RoboDK station: kr30 cnc template amana 46348 - paulina NEW THING 2.rdk

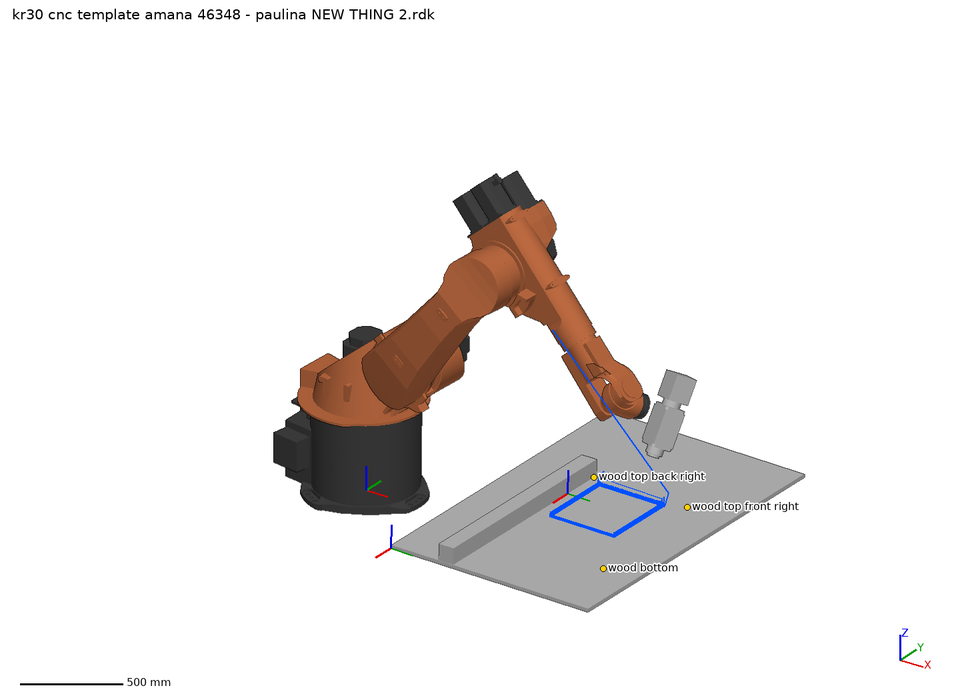
[picture v0: the station drawn from its stored meshes, robots at their saved joint values, targets as dots, program paths as lines]
Station kr30 cnc template amana 46348 - paulina NEW THING 2. Poses are relative to the parent item; angles as X-Y-Z fixed-axis rotations.
  - frame KUKA KR 30 HA Base at (0, 0, 0) mm
    - robot KUKA KR 30 HA: 6 axes, payload 30 kg, reach 2033 mm, repeatability 0.05 mm, weight 665 kg
        modified DH rows (alpha deg, a mm, theta deg, d mm): 0, 0, 0, 815; -90, 350, 0, 0; 0, 850, -90, 0; -90, 145, 0, 820; 90, 0, 0, 0; -90, 0, 180, 170
        joint limits [-185, -135, -120, -350, -119, -350] to [185, 35, 158, 350, 119, 350]; home [0, -90, 90, 0, 0, 0]; saved at [2.902, -51.207, 99.996, 272.3, 54.468, -220.075]
      - tool rc90 spindle mm, TCP at (267.95, 0.68, 160.99) mm, rotated rx 0 ry 90 rz 0 deg, size 110 x 421.3 x 118 mm, geometry from rc90 spindle mm.stl
    - frame Tabletop at (921.82, -1104.91, 385) mm, rotated rx -0.93 ry -0.21 rz -89.9 deg
      - object tabletop CHECK HEIGHT at (-1839.9, 0, 0) mm, size 1839.9 x 1168.4 x 19 mm, geometry from kr30 tabletop mm.stl
      - object kr30 pipe jig base at (-1220, -610.6, 0) mm, size 1217.6 x 88.9 x 88.9 mm, geometry from kr30 pipe jig base.stl
      - frame Frame 3 at (-930, 400, 45) mm
      - target wood top back right (Cartesian target) at (-1141.49, 406.84, 52.26) mm, rotated rx 18.07 ry 89.88 rz 108.17 deg; joints [-2.086, -55.392, 143.759, 178.106, 87.553, -179.775] of KUKA KR 30 HA
      - target wood bottom (Cartesian target) at (-376.62, 995.52, 35.89) mm, rotated rx 18.07 ry 89.88 rz 108.17 deg; joints [24.587, -27.296, 76.752, 211.623, 53.064, -199.759] of KUKA KR 30 HA
      - target wood top front right (Cartesian target) at (-1142.68, 960.22, 52.55) mm, rotated rx 18.06 ry 89.88 rz 108.16 deg; joints [-1.42, -37.516, 98.016, 178.579, 59.693, -179.129] of KUKA KR 30 HA
  - machining project Machining Settings: C:/Users/Research Office/Desktop/paulina a5.apt | rotZ(0) | rotX(0)*rotY(0) | rotZ(0)
  - program Machining (2349 instructions, listed below)
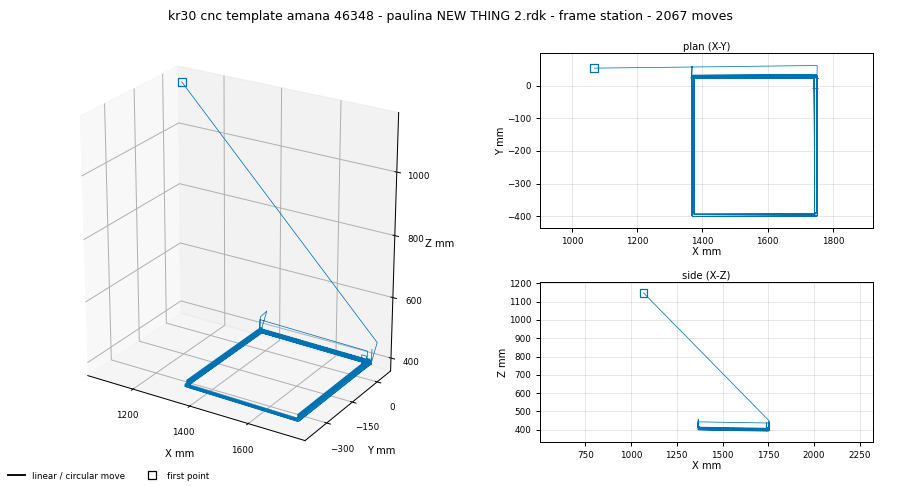
[picture p0: tool path of kr30 cnc template amana 46348 - paulina NEW THING 2.rdk in frame station, 2067 of 2067 moves have a stored position in this frame; points joined in program order, loops and branches not executed]

--- program Machining (robot KUKA KR 30 HA) ---
  Smooth(10)
  Print: /'1001'
  Print: /''
  Print: /'diagonal cut'
  Set speed (100.0 mm/s)
  Set Ref.: Frame 3
  Set Tool: rc90 spindle mm
  Show rc90 spindle mm
  MoveJ 1 to (-225.94, -263.82, 724.05) mm, rotated rx -179.73 ry 3.45 rz -91.41 deg; joints [-5.005, -121.314, 141.062, 163.754, 23.118, -164.211]
  MoveL 2 to (-235.36, 431, 39.15) mm, rotated rx -174.06 ry -29.54 rz -11.91 deg; joints [2.832, -37.469, 83.05, -73.25, 63.513, 134.274]
  MoveL 3 to (-235.36, 431, 39.15) mm, rotated rx -174.06 ry -29.54 rz -11.91 deg; joints [2.832, -37.469, 83.05, -73.25, 63.513, 134.274]
  Set speed (100.0 mm/s)
  MoveL 4 to (-206.65, 431, -10.41) mm, rotated rx -174.06 ry -29.54 rz -11.91 deg; joints [3.804, -35.34, 82.979, -73.62, 63.566, 136.691]
  Set speed (38.1 mm/s)
  MoveL 5 to (-201.55, 431, -19.21) mm, rotated rx -174.06 ry -29.54 rz -11.91 deg; joints [3.976, -34.949, 82.939, -73.676, 63.579, 137.104]
  MoveL 6 to (-200.68, 431, -19.44) mm, rotated rx -174.06 ry -29.54 rz -11.91 deg; joints [4.005, -34.936, 82.932, -73.66, 63.596, 137.117]
  Set speed (76.2 mm/s)
  MoveL 7 to (-202.44, 431, -12.48) mm, rotated rx -174.06 ry -29.54 rz -11.91 deg; joints [3.945, -35.237, 82.947, -73.562, 63.638, 136.796]
  MoveL 8 to (-201.13, 431, -12.23) mm, rotated rx -174.06 ry -29.54 rz -11.91 deg; joints [3.989, -35.243, 82.936, -73.526, 63.671, 136.788]
  MoveL 9 to (-196.56, 431, -16.91) mm, rotated rx -174.06 ry -29.54 rz -11.91 deg; joints [4.143, -35.027, 82.898, -73.511, 63.72, 137.012]
  Set speed (38.1 mm/s)
  MoveL 10 to (-196.33, 431, -16.04) mm, rotated rx -174.06 ry -29.54 rz -11.91 deg; joints [4.151, -35.063, 82.897, -73.488, 63.735, 136.973]
  Set speed (100.0 mm/s)
  MoveL 11 to (-203.65, 431, -3.41) mm, rotated rx -174.06 ry -29.54 rz -11.91 deg; joints [3.903, -35.623, 82.951, -73.408, 63.719, 136.379]
  MoveL 12 to (-199.05, 427.82, -0.75) mm, rotated rx -174.06 ry -29.54 rz -11.91 deg; joints [4.065, -35.896, 83.273, -73.328, 63.81, 136.466]
  Set speed (38.1 mm/s)
  MoveL 13 to (-197.47, 427.82, -3.47) mm, rotated rx -174.06 ry -29.54 rz -11.91 deg; joints [4.118, -35.776, 83.262, -73.346, 63.813, 136.595]
  MoveL 14 to (-197.39, 427.82, -3.84) mm, rotated rx -174.06 ry -29.54 rz -11.91 deg; joints [4.121, -35.76, 83.262, -73.351, 63.811, 136.612]
  Set speed (76.2 mm/s)
  MoveL 15 to (-197.71, 427.82, -8.22) mm, rotated rx -174.06 ry -29.54 rz -11.91 deg; joints [4.111, -35.578, 83.268, -73.446, 63.75, 136.812]
  MoveL 16 to (-199.91, 427.82, -8.42) mm, rotated rx -174.06 ry -29.54 rz -11.91 deg; joints [4.037, -35.578, 83.287, -73.503, 63.697, 136.816]
  MoveL 17 to (-206.05, 427.82, -11.57) mm, rotated rx -174.06 ry -29.54 rz -11.91 deg; joints [3.831, -35.468, 83.337, -73.712, 63.519, 136.944]
  MoveL 18 to (-201.08, 427.82, -20.25) mm, rotated rx -174.06 ry -29.54 rz -11.91 deg; joints [4, -35.081, 83.297, -73.769, 63.53, 137.352]
  MoveL 19 to (-201.08, 424.65, -20.25) mm, rotated rx -174.06 ry -29.54 rz -11.91 deg; joints [4.008, -35.258, 83.658, -73.852, 63.484, 137.55]
  MoveL 20 to (-206.05, 424.65, -11.57) mm, rotated rx -174.06 ry -29.54 rz -11.91 deg; joints [3.839, -35.646, 83.698, -73.795, 63.473, 137.141]
  MoveL 21 to (-200.05, 424.65, -8.41) mm, rotated rx -174.06 ry -29.54 rz -11.91 deg; joints [4.04, -35.757, 83.649, -73.588, 63.648, 137.012]
  MoveL 22 to (-197.85, 424.65, -8.4) mm, rotated rx -174.06 ry -29.54 rz -11.91 deg; joints [4.115, -35.749, 83.63, -73.535, 63.698, 137.016]
  MoveL 23 to (-197.85, 424.65, -4.14) mm, rotated rx -174.06 ry -29.54 rz -11.91 deg; joints [4.114, -35.928, 83.627, -73.449, 63.75, 136.821]
  Set speed (38.1 mm/s)
  MoveL 24 to (-197.89, 424.65, -3.98) mm, rotated rx -174.06 ry -29.54 rz -11.91 deg; joints [4.112, -35.935, 83.627, -73.446, 63.751, 136.814]
  MoveL 25 to (-198.05, 424.33, -3.7) mm, rotated rx -174.06 ry -29.54 rz -11.91 deg; joints [4.108, -35.965, 83.664, -73.453, 63.746, 136.82]
  Set speed (76.2 mm/s)
  MoveL 26 to (-198.05, 421.79, -3.7) mm, rotated rx -174.06 ry -29.54 rz -11.91 deg; joints [4.114, -36.107, 83.952, -73.517, 63.708, 136.976]
  Set speed (38.1 mm/s)
  MoveL 27 to (-197.89, 421.47, -3.98) mm, rotated rx -174.06 ry -29.54 rz -11.91 deg; joints [4.12, -36.113, 83.986, -73.527, 63.704, 137.009]
  MoveL 28 to (-197.85, 421.47, -4.14) mm, rotated rx -174.06 ry -29.54 rz -11.91 deg; joints [4.122, -36.106, 83.986, -73.529, 63.703, 137.017]
  Set speed (76.2 mm/s)
  MoveL 29 to (-197.85, 421.47, -8.28) mm, rotated rx -174.06 ry -29.54 rz -11.91 deg; joints [4.122, -35.931, 83.989, -73.613, 63.653, 137.207]
  MoveL 30 to (-200, 421.47, -8.41) mm, rotated rx -174.06 ry -29.54 rz -11.91 deg; joints [4.05, -35.934, 84.007, -73.668, 63.602, 137.208]
  MoveL 31 to (-206.05, 421.47, -11.57) mm, rotated rx -174.06 ry -29.54 rz -11.91 deg; joints [3.846, -35.823, 84.057, -73.878, 63.427, 137.338]
  MoveL 32 to (-201.08, 421.47, -20.25) mm, rotated rx -174.06 ry -29.54 rz -11.91 deg; joints [4.015, -35.434, 84.017, -73.934, 63.438, 137.748]
  MoveL 33 to (-201.08, 418.3, -20.25) mm, rotated rx -174.06 ry -29.54 rz -11.91 deg; joints [4.023, -35.609, 84.375, -74.017, 63.393, 137.946]
  MoveL 34 to (-206.05, 418.3, -11.57) mm, rotated rx -174.06 ry -29.54 rz -11.91 deg; joints [3.854, -35.999, 84.415, -73.96, 63.382, 137.535]
  MoveL 35 to (-199.95, 418.3, -8.41) mm, rotated rx -174.06 ry -29.54 rz -11.91 deg; joints [4.059, -36.111, 84.365, -73.748, 63.558, 137.404]
  MoveL 36 to (-197.85, 418.3, -8.16) mm, rotated rx -174.06 ry -29.54 rz -11.91 deg; joints [4.13, -36.113, 84.347, -73.692, 63.609, 137.397]
  MoveL 37 to (-197.85, 418.3, -4.14) mm, rotated rx -174.06 ry -29.54 rz -11.91 deg; joints [4.13, -36.283, 84.344, -73.61, 63.657, 137.211]
  Set speed (38.1 mm/s)
  MoveL 38 to (-197.89, 418.3, -3.98) mm, rotated rx -174.06 ry -29.54 rz -11.91 deg; joints [4.128, -36.29, 84.344, -73.608, 63.658, 137.204]
  MoveL 39 to (-198.05, 417.98, -3.7) mm, rotated rx -174.06 ry -29.54 rz -11.91 deg; joints [4.123, -36.32, 84.381, -73.614, 63.653, 137.21]
  Set speed (76.2 mm/s)
  MoveL 40 to (-198.05, 415.44, -3.7) mm, rotated rx -174.06 ry -29.54 rz -11.91 deg; joints [4.13, -36.461, 84.666, -73.678, 63.617, 137.366]
  Set speed (38.1 mm/s)
  MoveL 41 to (-197.89, 415.12, -3.98) mm, rotated rx -174.06 ry -29.54 rz -11.91 deg; joints [4.136, -36.467, 84.7, -73.688, 63.613, 137.398]
  MoveL 42 to (-197.85, 415.12, -4.14) mm, rotated rx -174.06 ry -29.54 rz -11.91 deg; joints [4.138, -36.46, 84.7, -73.69, 63.612, 137.406]
  Set speed (76.2 mm/s)
  MoveL 43 to (-197.85, 415.12, -8.4) mm, rotated rx -174.06 ry -29.54 rz -11.91 deg; joints [4.138, -36.279, 84.703, -73.778, 63.561, 137.603]
  MoveL 44 to (-199.9, 415.12, -8.41) mm, rotated rx -174.06 ry -29.54 rz -11.91 deg; joints [4.069, -36.286, 84.72, -73.828, 63.514, 137.599]
  MoveL 45 to (-206.05, 415.12, -11.57) mm, rotated rx -174.06 ry -29.54 rz -11.91 deg; joints [3.861, -36.175, 84.771, -74.042, 63.337, 137.73]
  MoveL 46 to (-201.08, 415.12, -20.25) mm, rotated rx -174.06 ry -29.54 rz -11.91 deg; joints [4.031, -35.784, 84.731, -74.099, 63.348, 138.142]
  MoveL 47 to (-201.08, 411.95, -20.25) mm, rotated rx -174.06 ry -29.54 rz -11.91 deg; joints [4.038, -35.958, 85.086, -74.181, 63.303, 138.338]
  MoveL 48 to (-206.05, 411.95, -11.57) mm, rotated rx -174.06 ry -29.54 rz -11.91 deg; joints [3.868, -36.35, 85.125, -74.124, 63.292, 137.925]
  MoveL 49 to (-199.84, 411.95, -8.41) mm, rotated rx -174.06 ry -29.54 rz -11.91 deg; joints [4.078, -36.461, 85.075, -73.907, 63.47, 137.793]
  MoveL 50 to (-197.85, 411.95, -8.4) mm, rotated rx -174.06 ry -29.54 rz -11.91 deg; joints [4.146, -36.454, 85.058, -73.858, 63.516, 137.798]
  MoveL 51 to (-197.85, 411.95, -4.14) mm, rotated rx -174.06 ry -29.54 rz -11.91 deg; joints [4.145, -36.635, 85.055, -73.77, 63.567, 137.599]
  Set speed (38.1 mm/s)
  MoveL 52 to (-197.89, 411.95, -3.98) mm, rotated rx -174.06 ry -29.54 rz -11.91 deg; joints [4.144, -36.642, 85.055, -73.768, 63.568, 137.592]
  MoveL 53 to (-198.05, 411.63, -3.7) mm, rotated rx -174.06 ry -29.54 rz -11.91 deg; joints [4.139, -36.672, 85.092, -73.774, 63.563, 137.598]
  Set speed (76.2 mm/s)
  MoveL 54 to (-198.05, 409.09, -3.7) mm, rotated rx -174.06 ry -29.54 rz -11.91 deg; joints [4.146, -36.812, 85.374, -73.838, 63.527, 137.752]
  Set speed (38.1 mm/s)
  MoveL 55 to (-197.89, 408.77, -3.98) mm, rotated rx -174.06 ry -29.54 rz -11.91 deg; joints [4.152, -36.817, 85.409, -73.848, 63.523, 137.785]
  MoveL 56 to (-197.85, 408.77, -4.14) mm, rotated rx -174.06 ry -29.54 rz -11.91 deg; joints [4.153, -36.81, 85.408, -73.85, 63.522, 137.792]
  Set speed (76.2 mm/s)
  MoveL 57 to (-197.85, 408.77, -8.4) mm, rotated rx -174.06 ry -29.54 rz -11.91 deg; joints [4.154, -36.629, 85.412, -73.939, 63.471, 137.991]
  MoveL 58 to (-200.19, 408.77, -8.41) mm, rotated rx -174.06 ry -29.54 rz -11.91 deg; joints [4.074, -36.637, 85.431, -73.996, 63.418, 137.986]
  MoveL 59 to (-206.05, 408.77, -11.57) mm, rotated rx -174.06 ry -29.54 rz -11.91 deg; joints [3.876, -36.524, 85.479, -74.206, 63.248, 138.12]
  MoveL 60 to (-201.08, 408.77, -20.25) mm, rotated rx -174.06 ry -29.54 rz -11.91 deg; joints [4.046, -36.132, 85.439, -74.263, 63.259, 138.534]
  MoveL 61 to (-201.08, 405.6, -20.25) mm, rotated rx -174.06 ry -29.54 rz -11.91 deg; joints [4.054, -36.304, 85.791, -74.345, 63.216, 138.729]
  MoveL 62 to (-206.05, 405.6, -11.57) mm, rotated rx -174.06 ry -29.54 rz -11.91 deg; joints [3.883, -36.697, 85.83, -74.287, 63.204, 138.313]
  MoveL 63 to (-200.12, 405.6, -8.41) mm, rotated rx -174.06 ry -29.54 rz -11.91 deg; joints [4.085, -36.811, 85.782, -74.075, 63.375, 138.179]
  MoveL 64 to (-197.85, 405.6, -8.4) mm, rotated rx -174.06 ry -29.54 rz -11.91 deg; joints [4.162, -36.802, 85.764, -74.019, 63.427, 138.184]
  MoveL 65 to (-197.85, 405.6, -4.14) mm, rotated rx -174.06 ry -29.54 rz -11.91 deg; joints [4.161, -36.985, 85.76, -73.93, 63.478, 137.985]
  MoveL 66 to (-197.85, 405.47, -3.66) mm, rotated rx -174.06 ry -29.54 rz -11.91 deg; joints [4.162, -37.012, 85.774, -73.923, 63.482, 137.97]
  MoveL 67 to (-197.85, 405.12, -3.31) mm, rotated rx -174.06 ry -29.54 rz -11.91 deg; joints [4.163, -37.046, 85.812, -73.925, 63.481, 137.975]
  MoveL 68 to (-197.85, 404.64, -3.19) mm, rotated rx -174.06 ry -29.54 rz -11.91 deg; joints [4.164, -37.078, 85.865, -73.934, 63.476, 137.998]
  MoveL 69 to (-197.85, 403.38, -3.19) mm, rotated rx -174.06 ry -29.54 rz -11.91 deg; joints [4.167, -37.147, 86.005, -73.966, 63.458, 138.074]
  MoveL 70 to (-197.85, 402.9, -3.31) mm, rotated rx -174.06 ry -29.54 rz -11.91 deg; joints [4.168, -37.168, 86.058, -73.981, 63.45, 138.109]
  MoveL 71 to (-197.85, 402.55, -3.66) mm, rotated rx -174.06 ry -29.54 rz -11.91 deg; joints [4.169, -37.172, 86.096, -73.997, 63.441, 138.146]
  MoveL 72 to (-197.85, 402.42, -4.14) mm, rotated rx -174.06 ry -29.54 rz -11.91 deg; joints [4.17, -37.158, 86.111, -74.01, 63.434, 138.176]
  MoveL 73 to (-197.85, 402.42, -8.4) mm, rotated rx -174.06 ry -29.54 rz -11.91 deg; joints [4.17, -36.976, 86.114, -74.099, 63.383, 138.376]
  MoveL 74 to (-200.05, 402.42, -8.41) mm, rotated rx -174.06 ry -29.54 rz -11.91 deg; joints [4.095, -36.984, 86.132, -74.154, 63.333, 138.372]
  MoveL 75 to (-206.05, 402.42, -11.57) mm, rotated rx -174.06 ry -29.54 rz -11.91 deg; joints [3.891, -36.87, 86.181, -74.369, 63.161, 138.507]
  MoveL 76 to (-201.08, 402.42, -20.25) mm, rotated rx -174.06 ry -29.54 rz -11.91 deg; joints [4.062, -36.476, 86.142, -74.427, 63.173, 138.923]
  MoveL 77 to (-201.08, 399.25, -20.25) mm, rotated rx -174.06 ry -29.54 rz -11.91 deg; joints [4.07, -36.647, 86.491, -74.508, 63.13, 139.117]
  MoveL 78 to (-206.05, 399.25, -11.57) mm, rotated rx -174.06 ry -29.54 rz -11.91 deg; joints [3.898, -37.042, 86.53, -74.45, 63.118, 138.699]
  MoveL 79 to (-199.98, 399.25, -8.41) mm, rotated rx -174.06 ry -29.54 rz -11.91 deg; joints [4.105, -37.156, 86.481, -74.232, 63.292, 138.564]
  MoveL 80 to (-197.85, 399.25, -8.4) mm, rotated rx -174.06 ry -29.54 rz -11.91 deg; joints [4.178, -37.148, 86.463, -74.179, 63.34, 138.568]
  MoveL 81 to (-197.85, 399.25, -4.14) mm, rotated rx -174.06 ry -29.54 rz -11.91 deg; joints [4.178, -37.331, 86.46, -74.089, 63.391, 138.368]
  Set speed (38.1 mm/s)
  MoveL 82 to (-197.89, 399.25, -3.98) mm, rotated rx -174.06 ry -29.54 rz -11.91 deg; joints [4.176, -37.338, 86.46, -74.087, 63.392, 138.36]
  MoveL 83 to (-198.05, 398.93, -3.7) mm, rotated rx -174.06 ry -29.54 rz -11.91 deg; joints [4.171, -37.368, 86.496, -74.093, 63.387, 138.366]
  Set speed (76.2 mm/s)
  MoveL 84 to (-198.05, 396.39, -3.7) mm, rotated rx -174.06 ry -29.54 rz -11.91 deg; joints [4.178, -37.506, 86.775, -74.156, 63.353, 138.518]
  Set speed (38.1 mm/s)
  MoveL 85 to (-197.89, 396.07, -3.98) mm, rotated rx -174.06 ry -29.54 rz -11.91 deg; joints [4.184, -37.511, 86.808, -74.166, 63.349, 138.55]
  MoveL 86 to (-197.85, 396.07, -4.14) mm, rotated rx -174.06 ry -29.54 rz -11.91 deg; joints [4.186, -37.504, 86.808, -74.169, 63.348, 138.558]
  Set speed (76.2 mm/s)
  MoveL 87 to (-197.85, 396.07, -8.4) mm, rotated rx -174.06 ry -29.54 rz -11.91 deg; joints [4.186, -37.32, 86.811, -74.258, 63.297, 138.759]
  MoveL 88 to (-199.91, 396.07, -8.41) mm, rotated rx -174.06 ry -29.54 rz -11.91 deg; joints [4.116, -37.328, 86.828, -74.31, 63.251, 138.756]
  MoveL 89 to (-206.05, 396.07, -11.57) mm, rotated rx -174.06 ry -29.54 rz -11.91 deg; joints [3.906, -37.214, 86.878, -74.531, 63.076, 138.891]
  MoveL 90 to (-201.08, 396.07, -20.25) mm, rotated rx -174.06 ry -29.54 rz -11.91 deg; joints [4.078, -36.818, 86.839, -74.589, 63.088, 139.31]
  MoveL 91 to (-201.08, 392.9, -20.25) mm, rotated rx -174.06 ry -29.54 rz -11.91 deg; joints [4.086, -36.988, 87.185, -74.671, 63.046, 139.502]
  MoveL 92 to (-206.05, 392.9, -11.57) mm, rotated rx -174.06 ry -29.54 rz -11.91 deg; joints [3.914, -37.384, 87.224, -74.612, 63.034, 139.083]
  MoveL 93 to (-199.84, 392.9, -8.41) mm, rotated rx -174.06 ry -29.54 rz -11.91 deg; joints [4.126, -37.498, 87.174, -74.388, 63.21, 138.946]
  MoveL 94 to (-197.85, 392.9, -8.38) mm, rotated rx -174.06 ry -29.54 rz -11.91 deg; joints [4.195, -37.492, 87.158, -74.337, 63.255, 138.949]
  MoveL 95 to (-197.85, 392.9, -4.14) mm, rotated rx -174.06 ry -29.54 rz -11.91 deg; joints [4.194, -37.675, 87.155, -74.248, 63.305, 138.748]
  Set speed (38.1 mm/s)
  MoveL 96 to (-197.89, 392.9, -3.98) mm, rotated rx -174.06 ry -29.54 rz -11.91 deg; joints [4.192, -37.682, 87.155, -74.245, 63.306, 138.74]
  MoveL 97 to (-198.05, 392.58, -3.7) mm, rotated rx -174.06 ry -29.54 rz -11.91 deg; joints [4.188, -37.712, 87.19, -74.251, 63.302, 138.746]
  Set speed (76.2 mm/s)
  MoveL 98 to (-198.05, 390.04, -3.7) mm, rotated rx -174.06 ry -29.54 rz -11.91 deg; joints [4.194, -37.849, 87.467, -74.315, 63.268, 138.898]
  Set speed (38.1 mm/s)
  MoveL 99 to (-197.89, 389.72, -3.98) mm, rotated rx -174.06 ry -29.54 rz -11.91 deg; joints [4.201, -37.853, 87.5, -74.324, 63.264, 138.93]
  MoveL 100 to (-197.85, 389.72, -4.14) mm, rotated rx -174.06 ry -29.54 rz -11.91 deg; joints [4.202, -37.846, 87.5, -74.327, 63.263, 138.938]
  Set speed (76.2 mm/s)
  MoveL 101 to (-197.85, 389.72, -8.26) mm, rotated rx -174.06 ry -29.54 rz -11.91 deg; joints [4.203, -37.668, 87.503, -74.414, 63.215, 139.134]
  MoveL 102 to (-199.77, 389.72, -8.41) mm, rotated rx -174.06 ry -29.54 rz -11.91 deg; joints [4.136, -37.669, 87.519, -74.466, 63.169, 139.137]
  MoveL 103 to (-206.05, 389.72, -11.57) mm, rotated rx -174.06 ry -29.54 rz -11.91 deg; joints [3.921, -37.554, 87.569, -74.693, 62.992, 139.273]
  MoveL 104 to (-201.08, 389.72, -20.25) mm, rotated rx -174.06 ry -29.54 rz -11.91 deg; joints [4.094, -37.157, 87.53, -74.752, 63.004, 139.694]
  MoveL 105 to (-201.08, 386.55, -20.25) mm, rotated rx -174.06 ry -29.54 rz -11.91 deg; joints [4.102, -37.326, 87.874, -74.832, 62.963, 139.885]
  MoveL 106 to (-206.05, 386.55, -11.57) mm, rotated rx -174.06 ry -29.54 rz -11.91 deg; joints [3.929, -37.724, 87.913, -74.774, 62.951, 139.464]
  MoveL 107 to (-199.7, 386.55, -8.41) mm, rotated rx -174.06 ry -29.54 rz -11.91 deg; joints [4.147, -37.838, 87.862, -74.544, 63.13, 139.326]
  MoveL 108 to (-197.85, 386.55, -8.41) mm, rotated rx -174.06 ry -29.54 rz -11.91 deg; joints [4.211, -37.831, 87.847, -74.497, 63.171, 139.33]
  MoveL 109 to (-197.85, 386.55, -4.14) mm, rotated rx -174.06 ry -29.54 rz -11.91 deg; joints [4.21, -38.016, 87.844, -74.405, 63.221, 139.126]
  Set speed (38.1 mm/s)
  MoveL 110 to (-197.89, 386.55, -3.98) mm, rotated rx -174.06 ry -29.54 rz -11.91 deg; joints [4.209, -38.023, 87.844, -74.403, 63.222, 139.119]
  MoveL 111 to (-198.05, 386.23, -3.7) mm, rotated rx -174.06 ry -29.54 rz -11.91 deg; joints [4.204, -38.053, 87.879, -74.409, 63.218, 139.124]
  Set speed (76.2 mm/s)
  MoveL 112 to (-198.05, 383.69, -3.7) mm, rotated rx -174.06 ry -29.54 rz -11.91 deg; joints [4.211, -38.189, 88.153, -74.472, 63.185, 139.275]
  Set speed (38.1 mm/s)
  MoveL 113 to (-197.89, 383.37, -3.98) mm, rotated rx -174.06 ry -29.54 rz -11.91 deg; joints [4.217, -38.193, 88.187, -74.482, 63.181, 139.307]
  MoveL 114 to (-197.85, 383.37, -4.14) mm, rotated rx -174.06 ry -29.54 rz -11.91 deg; joints [4.219, -38.186, 88.186, -74.484, 63.18, 139.315]
  Set speed (76.2 mm/s)
  MoveL 115 to (-197.85, 383.37, -8.4) mm, rotated rx -174.06 ry -29.54 rz -11.91 deg; joints [4.219, -38.001, 88.19, -74.576, 63.13, 139.519]
  MoveL 116 to (-199.66, 383.37, -8.41) mm, rotated rx -174.06 ry -29.54 rz -11.91 deg; joints [4.157, -38.007, 88.204, -74.622, 63.09, 139.515]
  MoveL 117 to (-206.05, 383.37, -11.57) mm, rotated rx -174.06 ry -29.54 rz -11.91 deg; joints [3.937, -37.893, 88.256, -74.854, 62.91, 139.653]
  MoveL 118 to (-201.08, 383.37, -20.25) mm, rotated rx -174.06 ry -29.54 rz -11.91 deg; joints [4.11, -37.494, 88.217, -74.913, 62.922, 140.076]
  MoveL 119 to (-201.08, 380.2, -20.25) mm, rotated rx -174.06 ry -29.54 rz -11.91 deg; joints [4.118, -37.661, 88.558, -74.993, 62.882, 140.267]
  MoveL 120 to (-206.05, 380.2, -11.57) mm, rotated rx -174.06 ry -29.54 rz -11.91 deg; joints [3.944, -38.061, 88.597, -74.934, 62.87, 139.843]
  MoveL 121 to (-200.12, 380.2, -8.41) mm, rotated rx -174.06 ry -29.54 rz -11.91 deg; joints [4.149, -38.177, 88.549, -74.713, 63.039, 139.703]
  MoveL 122 to (-197.85, 380.2, -8.4) mm, rotated rx -174.06 ry -29.54 rz -11.91 deg; joints [4.228, -38.169, 88.531, -74.654, 63.09, 139.707]
  MoveL 123 to (-197.85, 380.2, -4.14) mm, rotated rx -174.06 ry -29.54 rz -11.91 deg; joints [4.227, -38.355, 88.528, -74.562, 63.139, 139.502]
  Set speed (38.1 mm/s)
  MoveL 124 to (-197.89, 380.2, -3.98) mm, rotated rx -174.06 ry -29.54 rz -11.91 deg; joints [4.225, -38.362, 88.528, -74.56, 63.14, 139.495]
  MoveL 125 to (-198.05, 379.88, -3.7) mm, rotated rx -174.06 ry -29.54 rz -11.91 deg; joints [4.221, -38.392, 88.563, -74.566, 63.136, 139.5]
  Set speed (76.2 mm/s)
  MoveL 126 to (-198.05, 377.34, -3.7) mm, rotated rx -174.06 ry -29.54 rz -11.91 deg; joints [4.227, -38.526, 88.835, -74.629, 63.103, 139.65]
  Set speed (38.1 mm/s)
  MoveL 127 to (-197.89, 377.02, -3.98) mm, rotated rx -174.06 ry -29.54 rz -11.91 deg; joints [4.234, -38.531, 88.868, -74.638, 63.1, 139.682]
  MoveL 128 to (-197.85, 377.02, -4.14) mm, rotated rx -174.06 ry -29.54 rz -11.91 deg; joints [4.235, -38.524, 88.868, -74.641, 63.099, 139.69]
  Set speed (76.2 mm/s)
  MoveL 129 to (-197.85, 377.02, -8.4) mm, rotated rx -174.06 ry -29.54 rz -11.91 deg; joints [4.236, -38.337, 88.871, -74.733, 63.049, 139.895]
  MoveL 130 to (-200.07, 377.02, -8.41) mm, rotated rx -174.06 ry -29.54 rz -11.91 deg; joints [4.159, -38.345, 88.889, -74.791, 62.999, 139.891]
  MoveL 131 to (-206.05, 377.02, -11.57) mm, rotated rx -174.06 ry -29.54 rz -11.91 deg; joints [3.952, -38.228, 88.937, -75.014, 62.83, 140.031]
  MoveL 132 to (-201.08, 377.02, -20.25) mm, rotated rx -174.06 ry -29.54 rz -11.91 deg; joints [4.126, -37.827, 88.898, -75.074, 62.842, 140.456]
  MoveL 133 to (-201.08, 373.85, -20.25) mm, rotated rx -174.06 ry -29.54 rz -11.91 deg; joints [4.134, -37.994, 89.237, -75.154, 62.803, 140.646]
  MoveL 134 to (-206.05, 373.85, -11.57) mm, rotated rx -174.06 ry -29.54 rz -11.91 deg; joints [3.96, -38.395, 89.276, -75.094, 62.79, 140.219]
  MoveL 135 to (-200.58, 373.85, -8.41) mm, rotated rx -174.06 ry -29.54 rz -11.91 deg; joints [4.149, -38.514, 89.232, -74.883, 62.948, 140.077]
  MoveL 136 to (-197.85, 373.85, -8.4) mm, rotated rx -174.06 ry -29.54 rz -11.91 deg; joints [4.244, -38.505, 89.21, -74.811, 63.009, 140.082]
  MoveL 137 to (-197.85, 373.85, -4.14) mm, rotated rx -174.06 ry -29.54 rz -11.91 deg; joints [4.243, -38.691, 89.207, -74.719, 63.059, 139.876]
  Set speed (38.1 mm/s)
  MoveL 138 to (-197.89, 373.85, -3.98) mm, rotated rx -174.06 ry -29.54 rz -11.91 deg; joints [4.242, -38.698, 89.207, -74.716, 63.06, 139.868]
  MoveL 139 to (-198.05, 373.53, -3.7) mm, rotated rx -174.06 ry -29.54 rz -11.91 deg; joints [4.237, -38.728, 89.242, -74.722, 63.055, 139.874]
  Set speed (76.2 mm/s)
  MoveL 140 to (-198.05, 370.99, -3.7) mm, rotated rx -174.06 ry -29.54 rz -11.91 deg; joints [4.244, -38.862, 89.512, -74.785, 63.023, 140.022]
  Set speed (38.1 mm/s)
  MoveL 141 to (-197.89, 370.68, -3.98) mm, rotated rx -174.06 ry -29.54 rz -11.91 deg; joints [4.25, -38.866, 89.545, -74.794, 63.02, 140.055]
  MoveL 142 to (-197.85, 370.68, -4.14) mm, rotated rx -174.06 ry -29.54 rz -11.91 deg; joints [4.252, -38.859, 89.545, -74.797, 63.019, 140.062]
  Set speed (76.2 mm/s)
  MoveL 143 to (-197.85, 370.68, -8.4) mm, rotated rx -174.06 ry -29.54 rz -11.91 deg; joints [4.253, -38.671, 89.548, -74.89, 62.97, 140.269]
  MoveL 144 to (-200.55, 370.67, -8.41) mm, rotated rx -174.06 ry -29.54 rz -11.91 deg; joints [4.159, -38.681, 89.569, -74.961, 62.909, 140.264]
  MoveL 145 to (-206.05, 370.68, -11.57) mm, rotated rx -174.06 ry -29.54 rz -11.91 deg; joints [3.968, -38.562, 89.613, -75.174, 62.751, 140.407]
  MoveL 146 to (-201.08, 370.68, -20.25) mm, rotated rx -174.06 ry -29.54 rz -11.91 deg; joints [4.142, -38.159, 89.575, -75.234, 62.764, 140.834]
  MoveL 147 to (-201.08, 367.5, -20.25) mm, rotated rx -174.06 ry -29.54 rz -11.91 deg; joints [4.15, -38.324, 89.911, -75.313, 62.725, 141.022]
  MoveL 148 to (-206.05, 367.5, -11.57) mm, rotated rx -174.06 ry -29.54 rz -11.91 deg; joints [3.976, -38.727, 89.95, -75.254, 62.712, 140.594]
  MoveL 149 to (-200.51, 367.5, -8.41) mm, rotated rx -174.06 ry -29.54 rz -11.91 deg; joints [4.168, -38.847, 89.906, -75.038, 62.871, 140.451]
  MoveL 150 to (-197.85, 367.5, -8.4) mm, rotated rx -174.06 ry -29.54 rz -11.91 deg; joints [4.261, -38.838, 89.884, -74.968, 62.93, 140.455]
  MoveL 151 to (-197.85, 367.5, -4.14) mm, rotated rx -174.06 ry -29.54 rz -11.91 deg; joints [4.26, -39.025, 89.881, -74.874, 62.98, 140.248]
  MoveL 152 to (-197.85, 367.37, -3.66) mm, rotated rx -174.06 ry -29.54 rz -11.91 deg; joints [4.26, -39.053, 89.894, -74.867, 62.984, 140.232]
  MoveL 153 to (-197.85, 367.02, -3.31) mm, rotated rx -174.06 ry -29.54 rz -11.91 deg; joints [4.261, -39.086, 89.931, -74.868, 62.983, 140.236]
  MoveL 154 to (-197.85, 366.55, -3.19) mm, rotated rx -174.06 ry -29.54 rz -11.91 deg; joints [4.263, -39.117, 89.981, -74.877, 62.979, 140.257]
  MoveL 155 to (-197.85, 365.28, -3.19) mm, rotated rx -174.06 ry -29.54 rz -11.91 deg; joints [4.266, -39.183, 90.115, -74.908, 62.963, 140.331]
  MoveL 156 to (-197.85, 364.8, -3.31) mm, rotated rx -174.06 ry -29.54 rz -11.91 deg; joints [4.267, -39.203, 90.165, -74.922, 62.956, 140.365]
  MoveL 157 to (-197.85, 364.45, -3.66) mm, rotated rx -174.06 ry -29.54 rz -11.91 deg; joints [4.268, -39.206, 90.202, -74.938, 62.948, 140.402]
  MoveL 158 to (-197.85, 364.33, -4.14) mm, rotated rx -174.06 ry -29.54 rz -11.91 deg; joints [4.269, -39.191, 90.216, -74.952, 62.941, 140.433]
  MoveL 159 to (-197.85, 364.33, -8.4) mm, rotated rx -174.06 ry -29.54 rz -11.91 deg; joints [4.269, -39.003, 90.22, -75.046, 62.892, 140.641]
  MoveL 160 to (-200.48, 364.33, -8.41) mm, rotated rx -174.06 ry -29.54 rz -11.91 deg; joints [4.178, -39.012, 90.241, -75.116, 62.833, 140.637]
  MoveL 161 to (-206.05, 364.33, -11.57) mm, rotated rx -174.06 ry -29.54 rz -11.91 deg; joints [3.984, -38.893, 90.285, -75.333, 62.674, 140.781]
  MoveL 162 to (-201.08, 364.33, -20.25) mm, rotated rx -174.06 ry -29.54 rz -11.91 deg; joints [4.159, -38.488, 90.246, -75.393, 62.687, 141.21]
  MoveL 163 to (-201.08, 361.15, -20.25) mm, rotated rx -174.06 ry -29.54 rz -11.91 deg; joints [4.167, -38.652, 90.581, -75.472, 62.649, 141.397]
  MoveL 164 to (-206.05, 361.15, -11.57) mm, rotated rx -174.06 ry -29.54 rz -11.91 deg; joints [3.991, -39.057, 90.619, -75.412, 62.636, 140.967]
  MoveL 165 to (-200.44, 361.15, -8.41) mm, rotated rx -174.06 ry -29.54 rz -11.91 deg; joints [4.187, -39.177, 90.574, -75.193, 62.796, 140.822]
  MoveL 166 to (-197.85, 361.15, -8.4) mm, rotated rx -174.06 ry -29.54 rz -11.91 deg; joints [4.278, -39.168, 90.554, -75.124, 62.853, 140.826]
  MoveL 167 to (-197.85, 361.15, -4.14) mm, rotated rx -174.06 ry -29.54 rz -11.91 deg; joints [4.277, -39.357, 90.551, -75.029, 62.902, 140.618]
  Set speed (38.1 mm/s)
  MoveL 168 to (-197.89, 361.15, -3.98) mm, rotated rx -174.06 ry -29.54 rz -11.91 deg; joints [4.276, -39.364, 90.551, -75.027, 62.903, 140.61]
  MoveL 169 to (-198.05, 360.83, -3.7) mm, rotated rx -174.06 ry -29.54 rz -11.91 deg; joints [4.271, -39.393, 90.585, -75.033, 62.899, 140.615]
  Set speed (76.2 mm/s)
  MoveL 170 to (-198.05, 358.29, -3.7) mm, rotated rx -174.06 ry -29.54 rz -11.91 deg; joints [4.278, -39.525, 90.852, -75.095, 62.868, 140.762]
  Set speed (38.1 mm/s)
  MoveL 171 to (-197.89, 357.98, -3.98) mm, rotated rx -174.06 ry -29.54 rz -11.91 deg; joints [4.284, -39.529, 90.884, -75.104, 62.865, 140.794]
  MoveL 172 to (-197.85, 357.98, -4.14) mm, rotated rx -174.06 ry -29.54 rz -11.91 deg; joints [4.286, -39.522, 90.884, -75.107, 62.864, 140.802]
  Set speed (76.2 mm/s)
  MoveL 173 to (-197.85, 357.98, -8.25) mm, rotated rx -174.06 ry -29.54 rz -11.91 deg; joints [4.286, -39.339, 90.887, -75.198, 62.817, 141.003]
  MoveL 174 to (-200.41, 357.98, -8.41) mm, rotated rx -174.06 ry -29.54 rz -11.91 deg; joints [4.197, -39.342, 90.907, -75.27, 62.758, 141.007]
  MoveL 175 to (-206.05, 357.98, -11.57) mm, rotated rx -174.06 ry -29.54 rz -11.91 deg; joints [3.999, -39.221, 90.952, -75.491, 62.598, 141.152]
  MoveL 176 to (-201.08, 357.98, -20.25) mm, rotated rx -174.06 ry -29.54 rz -11.91 deg; joints [4.175, -38.815, 90.914, -75.552, 62.611, 141.584]
  MoveL 177 to (-201.08, 354.8, -20.25) mm, rotated rx -174.06 ry -29.54 rz -11.91 deg; joints [4.183, -38.977, 91.245, -75.631, 62.574, 141.77]
  MoveL 178 to (-206.05, 354.8, -11.57) mm, rotated rx -174.06 ry -29.54 rz -11.91 deg; joints [4.007, -39.385, 91.284, -75.57, 62.561, 141.337]
  MoveL 179 to (-200.37, 354.8, -8.41) mm, rotated rx -174.06 ry -29.54 rz -11.91 deg; joints [4.206, -39.505, 91.239, -75.347, 62.721, 141.191]
  MoveL 180 to (-197.85, 354.8, -8.13) mm, rotated rx -174.06 ry -29.54 rz -11.91 deg; joints [4.295, -39.508, 91.219, -75.273, 62.781, 141.182]
  MoveL 181 to (-197.85, 354.8, -4.14) mm, rotated rx -174.06 ry -29.54 rz -11.91 deg; joints [4.294, -39.686, 91.215, -75.184, 62.826, 140.985]
  MoveL 182 to (-197.85, 354.67, -3.66) mm, rotated rx -174.06 ry -29.54 rz -11.91 deg; joints [4.294, -39.714, 91.228, -75.176, 62.83, 140.969]
  MoveL 183 to (-197.85, 354.33, -3.31) mm, rotated rx -174.06 ry -29.54 rz -11.91 deg; joints [4.295, -39.747, 91.264, -75.177, 62.83, 140.972]
  MoveL 184 to (-197.85, 353.85, -3.19) mm, rotated rx -174.06 ry -29.54 rz -11.91 deg; joints [4.297, -39.777, 91.314, -75.186, 62.826, 140.993]
  MoveL 185 to (-197.85, 352.58, -3.19) mm, rotated rx -174.06 ry -29.54 rz -11.91 deg; joints [4.3, -39.843, 91.446, -75.216, 62.811, 141.066]
  MoveL 186 to (-197.85, 352.1, -3.31) mm, rotated rx -174.06 ry -29.54 rz -11.91 deg; joints [4.301, -39.862, 91.496, -75.231, 62.804, 141.1]
  MoveL 187 to (-197.85, 351.75, -3.66) mm, rotated rx -174.06 ry -29.54 rz -11.91 deg; joints [4.302, -39.864, 91.532, -75.247, 62.796, 141.138]
  MoveL 188 to (-197.85, 351.63, -4.14) mm, rotated rx -174.06 ry -29.54 rz -11.91 deg; joints [4.303, -39.85, 91.546, -75.261, 62.789, 141.168]
  MoveL 189 to (-197.85, 351.63, -8.4) mm, rotated rx -174.06 ry -29.54 rz -11.91 deg; joints [4.303, -39.659, 91.549, -75.357, 62.74, 141.379]
  MoveL 190 to (-200.34, 351.63, -8.41) mm, rotated rx -174.06 ry -29.54 rz -11.91 deg; joints [4.216, -39.668, 91.569, -75.424, 62.685, 141.375]
  MoveL 191 to (-206.05, 351.63, -11.57) mm, rotated rx -174.06 ry -29.54 rz -11.91 deg; joints [4.015, -39.547, 91.614, -75.649, 62.524, 141.522]
  MoveL 192 to (-201.08, 351.63, -20.25) mm, rotated rx -174.06 ry -29.54 rz -11.91 deg; joints [4.192, -39.139, 91.576, -75.71, 62.537, 141.956]
  MoveL 193 to (-201.08, 348.45, -20.25) mm, rotated rx -174.06 ry -29.54 rz -11.91 deg; joints [4.2, -39.301, 91.906, -75.789, 62.501, 142.141]
  MoveL 194 to (-206.05, 348.45, -11.57) mm, rotated rx -174.06 ry -29.54 rz -11.91 deg; joints [4.023, -39.71, 91.944, -75.728, 62.488, 141.706]
  MoveL 195 to (-199.95, 348.45, -8.41) mm, rotated rx -174.06 ry -29.54 rz -11.91 deg; joints [4.238, -39.83, 91.896, -75.491, 62.657, 141.559]
  MoveL 196 to (-197.85, 348.45, -8.4) mm, rotated rx -174.06 ry -29.54 rz -11.91 deg; joints [4.312, -39.822, 91.879, -75.434, 62.703, 141.562]
  MoveL 197 to (-197.85, 348.45, -4.14) mm, rotated rx -174.06 ry -29.54 rz -11.91 deg; joints [4.311, -40.013, 91.876, -75.338, 62.752, 141.351]
  MoveL 198 to (-197.85, 348.32, -3.66) mm, rotated rx -174.06 ry -29.54 rz -11.91 deg; joints [4.312, -40.041, 91.889, -75.33, 62.756, 141.335]
  MoveL 199 to (-197.85, 347.98, -3.31) mm, rotated rx -174.06 ry -29.54 rz -11.91 deg; joints [4.312, -40.074, 91.924, -75.33, 62.756, 141.337]
  MoveL 200 to (-197.85, 347.5, -3.19) mm, rotated rx -174.06 ry -29.54 rz -11.91 deg; joints [4.314, -40.104, 91.974, -75.339, 62.751, 141.358]
  MoveL 201 to (-197.85, 346.23, -3.19) mm, rotated rx -174.06 ry -29.54 rz -11.91 deg; joints [4.317, -40.169, 92.105, -75.37, 62.737, 141.431]
  MoveL 202 to (-197.85, 345.75, -3.31) mm, rotated rx -174.06 ry -29.54 rz -11.91 deg; joints [4.318, -40.188, 92.154, -75.384, 62.73, 141.465]
  MoveL 203 to (-197.85, 345.4, -3.66) mm, rotated rx -174.06 ry -29.54 rz -11.91 deg; joints [4.319, -40.19, 92.191, -75.4, 62.722, 141.502]
  MoveL 204 to (-197.85, 345.28, -4.14) mm, rotated rx -174.06 ry -29.54 rz -11.91 deg; joints [4.32, -40.175, 92.204, -75.414, 62.715, 141.533]
  MoveL 205 to (-197.85, 345.28, -8.4) mm, rotated rx -174.06 ry -29.54 rz -11.91 deg; joints [4.321, -39.984, 92.208, -75.511, 62.667, 141.745]
  MoveL 206 to (-199.91, 345.28, -8.41) mm, rotated rx -174.06 ry -29.54 rz -11.91 deg; joints [4.248, -39.992, 92.224, -75.567, 62.621, 141.742]
  MoveL 207 to (-206.05, 345.28, -11.57) mm, rotated rx -174.06 ry -29.54 rz -11.91 deg; joints [4.031, -39.872, 92.272, -75.806, 62.451, 141.889]
  MoveL 208 to (-201.08, 345.28, -20.25) mm, rotated rx -174.06 ry -29.54 rz -11.91 deg; joints [4.209, -39.461, 92.234, -75.867, 62.465, 142.326]
  MoveL 209 to (-201.08, 342.1, -20.25) mm, rotated rx -174.06 ry -29.54 rz -11.91 deg; joints [4.217, -39.622, 92.562, -75.946, 62.429, 142.51]
  MoveL 210 to (-206.05, 342.1, -11.57) mm, rotated rx -174.06 ry -29.54 rz -11.91 deg; joints [4.04, -40.033, 92.6, -75.884, 62.415, 142.072]
  MoveL 211 to (-199.87, 342.1, -8.41) mm, rotated rx -174.06 ry -29.54 rz -11.91 deg; joints [4.258, -40.153, 92.551, -75.643, 62.586, 141.925]
  MoveL 212 to (-197.85, 342.1, -8.4) mm, rotated rx -174.06 ry -29.54 rz -11.91 deg; joints [4.329, -40.146, 92.535, -75.588, 62.63, 141.927]
  MoveL 213 to (-197.85, 342.1, -4.14) mm, rotated rx -174.06 ry -29.54 rz -11.91 deg; joints [4.329, -40.338, 92.532, -75.491, 62.678, 141.715]
  Set speed (38.1 mm/s)
  MoveL 214 to (-197.89, 342.1, -3.98) mm, rotated rx -174.06 ry -29.54 rz -11.91 deg; joints [4.327, -40.345, 92.532, -75.488, 62.679, 141.707]
  MoveL 215 to (-198.05, 341.78, -3.7) mm, rotated rx -174.06 ry -29.54 rz -11.91 deg; joints [4.322, -40.374, 92.566, -75.494, 62.675, 141.711]
  Set speed (76.2 mm/s)
  MoveL 216 to (-198.05, 339.25, -3.7) mm, rotated rx -174.06 ry -29.54 rz -11.91 deg; joints [4.329, -40.503, 92.827, -75.555, 62.647, 141.856]
  Set speed (38.1 mm/s)
  MoveL 217 to (-197.89, 338.93, -3.98) mm, rotated rx -174.06 ry -29.54 rz -11.91 deg; joints [4.336, -40.506, 92.858, -75.565, 62.643, 141.888]
  MoveL 218 to (-197.85, 338.93, -4.14) mm, rotated rx -174.06 ry -29.54 rz -11.91 deg; joints [4.337, -40.499, 92.858, -75.567, 62.642, 141.896]
  Set speed (76.2 mm/s)
  MoveL 219 to (-197.85, 338.93, -8.4) mm, rotated rx -174.06 ry -29.54 rz -11.91 deg; joints [4.338, -40.307, 92.862, -75.664, 62.594, 142.109]
  MoveL 220 to (-200.2, 338.93, -8.41) mm, rotated rx -174.06 ry -29.54 rz -11.91 deg; joints [4.254, -40.315, 92.88, -75.729, 62.543, 142.106]
  MoveL 221 to (-206.05, 338.93, -11.57) mm, rotated rx -174.06 ry -29.54 rz -11.91 deg; joints [4.048, -40.193, 92.926, -75.963, 62.38, 142.255]
  MoveL 222 to (-201.08, 338.93, -20.25) mm, rotated rx -174.06 ry -29.54 rz -11.91 deg; joints [4.225, -39.781, 92.888, -76.024, 62.393, 142.694]
  MoveL 223 to (-201.08, 335.75, -20.25) mm, rotated rx -174.06 ry -29.54 rz -11.91 deg; joints [4.234, -39.941, 93.213, -76.102, 62.358, 142.877]
  MoveL 224 to (-206.05, 335.75, -11.57) mm, rotated rx -174.06 ry -29.54 rz -11.91 deg; joints [4.056, -40.354, 93.251, -76.041, 62.345, 142.437]
  MoveL 225 to (-200.15, 335.75, -8.41) mm, rotated rx -174.06 ry -29.54 rz -11.91 deg; joints [4.265, -40.476, 93.205, -75.805, 62.508, 142.288]
  MoveL 226 to (-197.85, 335.75, -8.4) mm, rotated rx -174.06 ry -29.54 rz -11.91 deg; joints [4.347, -40.468, 93.187, -75.741, 62.559, 142.29]
  MoveL 227 to (-197.85, 335.75, -4.14) mm, rotated rx -174.06 ry -29.54 rz -11.91 deg; joints [4.346, -40.66, 93.184, -75.643, 62.607, 142.077]
  Set speed (38.1 mm/s)
  MoveL 228 to (-197.89, 335.75, -3.98) mm, rotated rx -174.06 ry -29.54 rz -11.91 deg; joints [4.344, -40.667, 93.184, -75.641, 62.608, 142.069]
  MoveL 229 to (-198.05, 335.44, -3.7) mm, rotated rx -174.06 ry -29.54 rz -11.91 deg; joints [4.34, -40.697, 93.217, -75.646, 62.604, 142.073]
  Set speed (76.2 mm/s)
  MoveL 230 to (-198.05, 332.9, -3.7) mm, rotated rx -174.06 ry -29.54 rz -11.91 deg; joints [4.347, -40.825, 93.477, -75.707, 62.575, 142.217]
  Set speed (38.1 mm/s)
  MoveL 231 to (-197.89, 332.58, -3.98) mm, rotated rx -174.06 ry -29.54 rz -11.91 deg; joints [4.353, -40.828, 93.508, -75.717, 62.572, 142.249]
  MoveL 232 to (-197.85, 332.58, -4.14) mm, rotated rx -174.06 ry -29.54 rz -11.91 deg; joints [4.355, -40.821, 93.508, -75.719, 62.571, 142.257]
  Set speed (76.2 mm/s)
  MoveL 233 to (-197.85, 332.58, -8.4) mm, rotated rx -174.06 ry -29.54 rz -11.91 deg; joints [4.356, -40.628, 93.511, -75.817, 62.524, 142.471]
  MoveL 234 to (-200.15, 332.58, -8.41) mm, rotated rx -174.06 ry -29.54 rz -11.91 deg; joints [4.273, -40.636, 93.529, -75.882, 62.473, 142.469]
  MoveL 235 to (-206.05, 332.58, -11.57) mm, rotated rx -174.06 ry -29.54 rz -11.91 deg; joints [4.064, -40.513, 93.576, -76.118, 62.31, 142.619]
  MoveL 236 to (-201.08, 332.58, -20.25) mm, rotated rx -174.06 ry -29.54 rz -11.91 deg; joints [4.243, -40.099, 93.538, -76.18, 62.324, 143.06]
  MoveL 237 to (-201.08, 329.4, -20.25) mm, rotated rx -174.06 ry -29.54 rz -11.91 deg; joints [4.251, -40.257, 93.861, -76.258, 62.289, 143.243]
  MoveL 238 to (-206.05, 329.4, -11.57) mm, rotated rx -174.06 ry -29.54 rz -11.91 deg; joints [4.072, -40.672, 93.899, -76.196, 62.276, 142.8]
  MoveL 239 to (-200.15, 329.4, -8.41) mm, rotated rx -174.06 ry -29.54 rz -11.91 deg; joints [4.282, -40.795, 93.853, -75.958, 62.438, 142.649]
  MoveL 240 to (-197.85, 329.4, -8.4) mm, rotated rx -174.06 ry -29.54 rz -11.91 deg; joints [4.364, -40.787, 93.834, -75.894, 62.489, 142.652]
  MoveL 241 to (-197.85, 329.4, -4.14) mm, rotated rx -174.06 ry -29.54 rz -11.91 deg; joints [4.364, -40.981, 93.831, -75.795, 62.536, 142.437]
  Set speed (38.1 mm/s)
  MoveL 242 to (-197.89, 329.4, -3.98) mm, rotated rx -174.06 ry -29.54 rz -11.91 deg; joints [4.362, -40.988, 93.831, -75.793, 62.537, 142.429]
  MoveL 243 to (-198.05, 329.09, -3.7) mm, rotated rx -174.06 ry -29.54 rz -11.91 deg; joints [4.357, -41.017, 93.865, -75.798, 62.533, 142.432]
  Set speed (76.2 mm/s)
  MoveL 244 to (-198.05, 326.55, -3.7) mm, rotated rx -174.06 ry -29.54 rz -11.91 deg; joints [4.364, -41.145, 94.123, -75.859, 62.506, 142.576]
  Set speed (38.1 mm/s)
  MoveL 245 to (-197.89, 326.23, -3.98) mm, rotated rx -174.06 ry -29.54 rz -11.91 deg; joints [4.371, -41.148, 94.154, -75.868, 62.503, 142.608]
  MoveL 246 to (-197.85, 326.23, -4.14) mm, rotated rx -174.06 ry -29.54 rz -11.91 deg; joints [4.372, -41.14, 94.154, -75.871, 62.502, 142.616]
  Set speed (76.2 mm/s)
  MoveL 247 to (-197.85, 326.23, -8.4) mm, rotated rx -174.06 ry -29.54 rz -11.91 deg; joints [4.373, -40.946, 94.157, -75.97, 62.454, 142.832]
  MoveL 248 to (-200.15, 326.23, -8.41) mm, rotated rx -174.06 ry -29.54 rz -11.91 deg; joints [4.291, -40.954, 94.175, -76.035, 62.404, 142.829]
  MoveL 249 to (-206.05, 326.23, -11.57) mm, rotated rx -174.06 ry -29.54 rz -11.91 deg; joints [4.081, -40.831, 94.221, -76.274, 62.241, 142.981]
  MoveL 250 to (-201.08, 326.23, -20.25) mm, rotated rx -174.06 ry -29.54 rz -11.91 deg; joints [4.26, -40.415, 94.183, -76.336, 62.255, 143.425]
  MoveL 251 to (-201.08, 323.05, -20.25) mm, rotated rx -174.06 ry -29.54 rz -11.91 deg; joints [4.268, -40.572, 94.504, -76.414, 62.222, 143.606]
  MoveL 252 to (-206.05, 323.05, -11.57) mm, rotated rx -174.06 ry -29.54 rz -11.91 deg; joints [4.089, -40.989, 94.542, -76.351, 62.208, 143.162]
  MoveL 253 to (-200.15, 323.05, -8.41) mm, rotated rx -174.06 ry -29.54 rz -11.91 deg; joints [4.299, -41.113, 94.496, -76.111, 62.37, 143.009]
  MoveL 254 to (-197.85, 323.05, -8.4) mm, rotated rx -174.06 ry -29.54 rz -11.91 deg; joints [4.382, -41.105, 94.478, -76.046, 62.42, 143.011]
  MoveL 255 to (-197.85, 323.05, -4.14) mm, rotated rx -174.06 ry -29.54 rz -11.91 deg; joints [4.381, -41.299, 94.475, -75.946, 62.467, 142.795]
  Set speed (38.1 mm/s)
  MoveL 256 to (-197.89, 323.05, -3.98) mm, rotated rx -174.06 ry -29.54 rz -11.91 deg; joints [4.38, -41.307, 94.475, -75.944, 62.468, 142.787]
  MoveL 257 to (-198.05, 322.74, -3.7) mm, rotated rx -174.06 ry -29.54 rz -11.91 deg; joints [4.375, -41.336, 94.508, -75.949, 62.464, 142.79]
  Set speed (76.2 mm/s)
  MoveL 258 to (-198.05, 320.2, -3.7) mm, rotated rx -174.06 ry -29.54 rz -11.91 deg; joints [4.382, -41.462, 94.764, -76.01, 62.437, 142.933]
  Set speed (38.1 mm/s)
  MoveL 259 to (-197.89, 319.88, -3.98) mm, rotated rx -174.06 ry -29.54 rz -11.91 deg; joints [4.389, -41.465, 94.795, -76.019, 62.434, 142.965]
  MoveL 260 to (-197.85, 319.88, -4.14) mm, rotated rx -174.06 ry -29.54 rz -11.91 deg; joints [4.39, -41.458, 94.795, -76.022, 62.433, 142.973]
  Set speed (76.2 mm/s)
  MoveL 261 to (-197.85, 319.88, -8.4) mm, rotated rx -174.06 ry -29.54 rz -11.91 deg; joints [4.391, -41.263, 94.798, -76.122, 62.386, 143.191]
  MoveL 262 to (-200.15, 319.88, -8.41) mm, rotated rx -174.06 ry -29.54 rz -11.91 deg; joints [4.308, -41.271, 94.816, -76.187, 62.336, 143.188]
  MoveL 263 to (-206.05, 319.88, -11.57) mm, rotated rx -174.06 ry -29.54 rz -11.91 deg; joints [4.097, -41.147, 94.862, -76.428, 62.174, 143.342]
  MoveL 264 to (-201.08, 319.88, -20.25) mm, rotated rx -174.06 ry -29.54 rz -11.91 deg; joints [4.277, -40.729, 94.825, -76.491, 62.188, 143.788]
  MoveL 265 to (-201.08, 316.7, -20.25) mm, rotated rx -174.06 ry -29.54 rz -11.91 deg; joints [4.286, -40.885, 95.144, -76.568, 62.155, 143.968]
  MoveL 266 to (-206.05, 316.7, -11.57) mm, rotated rx -174.06 ry -29.54 rz -11.91 deg; joints [4.106, -41.304, 95.182, -76.506, 62.141, 143.521]
  MoveL 267 to (-200.15, 316.7, -8.41) mm, rotated rx -174.06 ry -29.54 rz -11.91 deg; joints [4.317, -41.428, 95.136, -76.263, 62.303, 143.367]
  MoveL 268 to (-197.85, 316.7, -8.4) mm, rotated rx -174.06 ry -29.54 rz -11.91 deg; joints [4.4, -41.42, 95.118, -76.197, 62.353, 143.369]
  MoveL 269 to (-197.85, 316.7, -4.14) mm, rotated rx -174.06 ry -29.54 rz -11.91 deg; joints [4.399, -41.616, 95.114, -76.097, 62.4, 143.151]
  Set speed (38.1 mm/s)
  MoveL 270 to (-197.89, 316.7, -3.98) mm, rotated rx -174.06 ry -29.54 rz -11.91 deg; joints [4.398, -41.623, 95.115, -76.094, 62.401, 143.143]
  MoveL 271 to (-198.05, 316.39, -3.7) mm, rotated rx -174.06 ry -29.54 rz -11.91 deg; joints [4.393, -41.652, 95.147, -76.1, 62.397, 143.147]
  Set speed (76.2 mm/s)
  MoveL 272 to (-198.05, 313.85, -3.7) mm, rotated rx -174.06 ry -29.54 rz -11.91 deg; joints [4.4, -41.778, 95.402, -76.16, 62.37, 143.289]
  Set speed (38.1 mm/s)
  MoveL 273 to (-197.89, 313.53, -3.98) mm, rotated rx -174.06 ry -29.54 rz -11.91 deg; joints [4.407, -41.781, 95.433, -76.17, 62.367, 143.321]
  MoveL 274 to (-197.85, 313.53, -4.14) mm, rotated rx -174.06 ry -29.54 rz -11.91 deg; joints [4.408, -41.773, 95.433, -76.172, 62.366, 143.329]
  Set speed (76.2 mm/s)
  MoveL 275 to (-197.85, 313.53, -8.4) mm, rotated rx -174.06 ry -29.54 rz -11.91 deg; joints [4.409, -41.577, 95.436, -76.273, 62.319, 143.548]
  MoveL 276 to (-200.15, 313.53, -8.41) mm, rotated rx -174.06 ry -29.54 rz -11.91 deg; joints [4.326, -41.585, 95.454, -76.339, 62.269, 143.545]
  MoveL 277 to (-206.05, 313.53, -11.57) mm, rotated rx -174.06 ry -29.54 rz -11.91 deg; joints [4.114, -41.46, 95.5, -76.582, 62.108, 143.7]
  MoveL 278 to (-201.08, 313.53, -20.25) mm, rotated rx -174.06 ry -29.54 rz -11.91 deg; joints [4.295, -41.04, 95.462, -76.646, 62.122, 144.149]
  MoveL 279 to (-201.08, 310.35, -20.25) mm, rotated rx -174.06 ry -29.54 rz -11.91 deg; joints [4.303, -41.196, 95.779, -76.723, 62.09, 144.329]
  MoveL 280 to (-206.05, 310.35, -11.57) mm, rotated rx -174.06 ry -29.54 rz -11.91 deg; joints [4.122, -41.616, 95.817, -76.659, 62.076, 143.879]
  MoveL 281 to (-200.15, 310.35, -8.41) mm, rotated rx -174.06 ry -29.54 rz -11.91 deg; joints [4.335, -41.742, 95.771, -76.415, 62.237, 143.723]
  MoveL 282 to (-197.85, 310.35, -8.4) mm, rotated rx -174.06 ry -29.54 rz -11.91 deg; joints [4.418, -41.734, 95.753, -76.348, 62.286, 143.725]
  MoveL 283 to (-197.85, 310.35, -4.14) mm, rotated rx -174.06 ry -29.54 rz -11.91 deg; joints [4.417, -41.93, 95.75, -76.247, 62.333, 143.506]
  Set speed (38.1 mm/s)
  MoveL 284 to (-197.89, 310.35, -3.98) mm, rotated rx -174.06 ry -29.54 rz -11.91 deg; joints [4.416, -41.938, 95.75, -76.244, 62.334, 143.498]
  MoveL 285 to (-198.05, 310.04, -3.7) mm, rotated rx -174.06 ry -29.54 rz -11.91 deg; joints [4.411, -41.967, 95.783, -76.25, 62.33, 143.501]
  Set speed (76.2 mm/s)
  MoveL 286 to (-198.05, 307.5, -3.7) mm, rotated rx -174.06 ry -29.54 rz -11.91 deg; joints [4.418, -42.092, 96.036, -76.31, 62.304, 143.643]
  Set speed (38.1 mm/s)
  MoveL 287 to (-197.89, 307.18, -3.98) mm, rotated rx -174.06 ry -29.54 rz -11.91 deg; joints [4.425, -42.094, 96.067, -76.319, 62.301, 143.675]
  MoveL 288 to (-197.85, 307.18, -4.14) mm, rotated rx -174.06 ry -29.54 rz -11.91 deg; joints [4.426, -42.087, 96.066, -76.322, 62.301, 143.683]
  Set speed (76.2 mm/s)
  MoveL 289 to (-197.85, 307.18, -8.4) mm, rotated rx -174.06 ry -29.54 rz -11.91 deg; joints [4.427, -41.89, 96.07, -76.424, 62.254, 143.903]
  MoveL 290 to (-200.15, 307.18, -8.41) mm, rotated rx -174.06 ry -29.54 rz -11.91 deg; joints [4.343, -41.898, 96.088, -76.49, 62.204, 143.901]
  MoveL 291 to (-206.05, 307.18, -11.57) mm, rotated rx -174.06 ry -29.54 rz -11.91 deg; joints [4.131, -41.772, 96.133, -76.736, 62.044, 144.057]
  MoveL 292 to (-201.08, 307.18, -20.25) mm, rotated rx -174.06 ry -29.54 rz -11.91 deg; joints [4.312, -41.35, 96.096, -76.8, 62.058, 144.508]
  MoveL 293 to (-201.08, 304.01, -20.25) mm, rotated rx -174.06 ry -29.54 rz -11.91 deg; joints [4.321, -41.504, 96.411, -76.876, 62.026, 144.687]
  MoveL 294 to (-206.05, 304.01, -11.57) mm, rotated rx -174.06 ry -29.54 rz -11.91 deg; joints [4.139, -41.927, 96.449, -76.813, 62.012, 144.235]
  MoveL 295 to (-200.15, 304.01, -8.41) mm, rotated rx -174.06 ry -29.54 rz -11.91 deg; joints [4.352, -42.054, 96.403, -76.566, 62.172, 144.078]
  MoveL 296 to (-197.85, 304.01, -8.4) mm, rotated rx -174.06 ry -29.54 rz -11.91 deg; joints [4.436, -42.046, 96.385, -76.499, 62.222, 144.08]
  MoveL 297 to (-197.85, 304.01, -4.14) mm, rotated rx -174.06 ry -29.54 rz -11.91 deg; joints [4.435, -42.243, 96.382, -76.396, 62.268, 143.859]
  Set speed (38.1 mm/s)
  MoveL 298 to (-197.89, 304.01, -3.98) mm, rotated rx -174.06 ry -29.54 rz -11.91 deg; joints [4.434, -42.251, 96.382, -76.394, 62.269, 143.851]
  MoveL 299 to (-198.05, 303.69, -3.7) mm, rotated rx -174.06 ry -29.54 rz -11.91 deg; joints [4.429, -42.279, 96.415, -76.399, 62.265, 143.854]
  Set speed (76.2 mm/s)
  MoveL 300 to (-198.05, 301.15, -3.7) mm, rotated rx -174.06 ry -29.54 rz -11.91 deg; joints [4.436, -42.404, 96.666, -76.459, 62.24, 143.995]
  Set speed (38.1 mm/s)
  MoveL 301 to (-197.89, 300.83, -3.98) mm, rotated rx -174.06 ry -29.54 rz -11.91 deg; joints [4.443, -42.406, 96.697, -76.468, 62.237, 144.027]
  MoveL 302 to (-197.85, 300.83, -4.14) mm, rotated rx -174.06 ry -29.54 rz -11.91 deg; joints [4.444, -42.399, 96.696, -76.471, 62.236, 144.035]
  Set speed (76.2 mm/s)
  MoveL 303 to (-197.85, 300.83, -8.4) mm, rotated rx -174.06 ry -29.54 rz -11.91 deg; joints [4.445, -42.201, 96.7, -76.574, 62.19, 144.257]
  MoveL 304 to (-200.15, 300.83, -8.41) mm, rotated rx -174.06 ry -29.54 rz -11.91 deg; joints [4.361, -42.209, 96.718, -76.641, 62.14, 144.255]
  MoveL 305 to (-206.05, 300.83, -11.57) mm, rotated rx -174.06 ry -29.54 rz -11.91 deg; joints [4.148, -42.082, 96.763, -76.889, 61.98, 144.413]
  MoveL 306 to (-201.08, 300.83, -20.25) mm, rotated rx -174.06 ry -29.54 rz -11.91 deg; joints [4.33, -41.658, 96.726, -76.953, 61.995, 144.866]
  MoveL 307 to (-201.08, 297.66, -20.25) mm, rotated rx -174.06 ry -29.54 rz -11.91 deg; joints [4.339, -41.811, 97.039, -77.029, 61.964, 145.044]
  MoveL 308 to (-206.05, 297.66, -11.57) mm, rotated rx -174.06 ry -29.54 rz -11.91 deg; joints [4.156, -42.236, 97.077, -76.965, 61.949, 144.59]
  MoveL 309 to (-200.15, 297.66, -8.41) mm, rotated rx -174.06 ry -29.54 rz -11.91 deg; joints [4.37, -42.363, 97.031, -76.716, 62.108, 144.431]
  MoveL 310 to (-197.85, 297.66, -8.4) mm, rotated rx -174.06 ry -29.54 rz -11.91 deg; joints [4.454, -42.355, 97.013, -76.648, 62.158, 144.433]
  MoveL 311 to (-197.85, 297.66, -4.14) mm, rotated rx -174.06 ry -29.54 rz -11.91 deg; joints [4.454, -42.554, 97.01, -76.545, 62.204, 144.211]
  Set speed (38.1 mm/s)
  MoveL 312 to (-197.89, 297.66, -3.98) mm, rotated rx -174.06 ry -29.54 rz -11.91 deg; joints [4.452, -42.561, 97.01, -76.543, 62.205, 144.202]
  MoveL 313 to (-198.05, 297.34, -3.7) mm, rotated rx -174.06 ry -29.54 rz -11.91 deg; joints [4.447, -42.59, 97.043, -76.548, 62.202, 144.205]
  Set speed (76.2 mm/s)
  MoveL 314 to (-198.05, 294.8, -3.7) mm, rotated rx -174.06 ry -29.54 rz -11.91 deg; joints [4.454, -42.714, 97.293, -76.608, 62.176, 144.346]
  Set speed (38.1 mm/s)
  MoveL 315 to (-197.89, 294.48, -3.98) mm, rotated rx -174.06 ry -29.54 rz -11.91 deg; joints [4.461, -42.716, 97.323, -76.617, 62.174, 144.378]
  MoveL 316 to (-197.85, 294.48, -4.14) mm, rotated rx -174.06 ry -29.54 rz -11.91 deg; joints [4.463, -42.709, 97.323, -76.62, 62.173, 144.386]
  Set speed (76.2 mm/s)
  MoveL 317 to (-197.85, 294.48, -8.4) mm, rotated rx -174.06 ry -29.54 rz -11.91 deg; joints [4.463, -42.51, 97.326, -76.723, 62.127, 144.609]
  MoveL 318 to (-200.15, 294.48, -8.41) mm, rotated rx -174.06 ry -29.54 rz -11.91 deg; joints [4.379, -42.518, 97.344, -76.791, 62.077, 144.607]
  MoveL 319 to (-206.05, 294.48, -11.57) mm, rotated rx -174.06 ry -29.54 rz -11.91 deg; joints [4.165, -42.39, 97.39, -77.041, 61.918, 144.766]
  MoveL 320 to (-201.08, 294.48, -20.25) mm, rotated rx -174.06 ry -29.54 rz -11.91 deg; joints [4.348, -41.964, 97.352, -77.106, 61.933, 145.222]
  MoveL 321 to (-201.08, 291.31, -20.25) mm, rotated rx -174.06 ry -29.54 rz -11.91 deg; joints [4.357, -42.116, 97.664, -77.182, 61.902, 145.4]
  MoveL 322 to (-206.05, 291.31, -11.57) mm, rotated rx -174.06 ry -29.54 rz -11.91 deg; joints [4.174, -42.544, 97.701, -77.117, 61.887, 144.943]
  MoveL 323 to (-200.15, 291.31, -8.41) mm, rotated rx -174.06 ry -29.54 rz -11.91 deg; joints [4.388, -42.671, 97.656, -76.866, 62.046, 144.783]
  MoveL 324 to (-197.85, 291.31, -8.4) mm, rotated rx -174.06 ry -29.54 rz -11.91 deg; joints [4.473, -42.663, 97.638, -76.798, 62.096, 144.784]
  MoveL 325 to (-197.85, 291.31, -4.14) mm, rotated rx -174.06 ry -29.54 rz -11.91 deg; joints [4.472, -42.863, 97.635, -76.694, 62.142, 144.561]
  Set speed (38.1 mm/s)
  MoveL 326 to (-197.89, 291.31, -3.98) mm, rotated rx -174.06 ry -29.54 rz -11.91 deg; joints [4.47, -42.871, 97.635, -76.691, 62.143, 144.552]
  MoveL 327 to (-198.05, 290.99, -3.7) mm, rotated rx -174.06 ry -29.54 rz -11.91 deg; joints [4.465, -42.899, 97.667, -76.696, 62.139, 144.555]
  Set speed (76.2 mm/s)
  MoveL 328 to (-198.05, 288.45, -3.7) mm, rotated rx -174.06 ry -29.54 rz -11.91 deg; joints [4.473, -43.023, 97.916, -76.756, 62.114, 144.695]
  Set speed (38.1 mm/s)
  MoveL 329 to (-197.89, 288.13, -3.98) mm, rotated rx -174.06 ry -29.54 rz -11.91 deg; joints [4.48, -43.024, 97.946, -76.765, 62.112, 144.727]
  MoveL 330 to (-197.85, 288.13, -4.14) mm, rotated rx -174.06 ry -29.54 rz -11.91 deg; joints [4.481, -43.017, 97.946, -76.768, 62.111, 144.735]
  Set speed (76.2 mm/s)
  MoveL 331 to (-197.85, 288.13, -8.4) mm, rotated rx -174.06 ry -29.54 rz -11.91 deg; joints [4.482, -42.817, 97.949, -76.872, 62.065, 144.959]
  MoveL 332 to (-200.15, 288.13, -8.41) mm, rotated rx -174.06 ry -29.54 rz -11.91 deg; joints [4.398, -42.825, 97.967, -76.94, 62.016, 144.958]
  MoveL 333 to (-206.05, 288.13, -11.57) mm, rotated rx -174.06 ry -29.54 rz -11.91 deg; joints [4.182, -42.696, 98.012, -77.193, 61.857, 145.119]
  MoveL 334 to (-201.08, 288.13, -20.25) mm, rotated rx -174.06 ry -29.54 rz -11.91 deg; joints [4.366, -42.268, 97.975, -77.258, 61.872, 145.577]
  MoveL 335 to (-201.08, 284.96, -20.25) mm, rotated rx -174.06 ry -29.54 rz -11.91 deg; joints [4.375, -42.42, 98.285, -77.334, 61.842, 145.754]
  MoveL 336 to (-206.05, 284.96, -11.57) mm, rotated rx -174.06 ry -29.54 rz -11.91 deg; joints [4.191, -42.849, 98.322, -77.269, 61.827, 145.294]
  MoveL 337 to (-200.15, 284.96, -8.41) mm, rotated rx -174.06 ry -29.54 rz -11.91 deg; joints [4.407, -42.978, 98.277, -77.015, 61.985, 145.132]
  MoveL 338 to (-197.85, 284.96, -8.4) mm, rotated rx -174.06 ry -29.54 rz -11.91 deg; joints [4.491, -42.97, 98.259, -76.946, 62.034, 145.134]
  MoveL 339 to (-197.85, 284.96, -4.14) mm, rotated rx -174.06 ry -29.54 rz -11.91 deg; joints [4.491, -43.17, 98.256, -76.841, 62.08, 144.909]
  Set speed (38.1 mm/s)
  MoveL 340 to (-197.89, 284.96, -3.98) mm, rotated rx -174.06 ry -29.54 rz -11.91 deg; joints [4.489, -43.178, 98.256, -76.839, 62.081, 144.9]
  MoveL 341 to (-198.05, 284.64, -3.7) mm, rotated rx -174.06 ry -29.54 rz -11.91 deg; joints [4.484, -43.207, 98.288, -76.844, 62.078, 144.903]
  Set speed (76.2 mm/s)
  MoveL 342 to (-198.05, 282.1, -3.7) mm, rotated rx -174.06 ry -29.54 rz -11.91 deg; joints [4.491, -43.329, 98.535, -76.903, 62.053, 145.042]
  Set speed (38.1 mm/s)
  MoveL 343 to (-197.89, 281.78, -3.98) mm, rotated rx -174.06 ry -29.54 rz -11.91 deg; joints [4.498, -43.331, 98.565, -76.912, 62.051, 145.074]
  MoveL 344 to (-197.85, 281.78, -4.14) mm, rotated rx -174.06 ry -29.54 rz -11.91 deg; joints [4.5, -43.323, 98.565, -76.915, 62.05, 145.082]
  Set speed (76.2 mm/s)
  MoveL 345 to (-197.85, 281.78, -8.4) mm, rotated rx -174.06 ry -29.54 rz -11.91 deg; joints [4.501, -43.122, 98.568, -77.02, 62.004, 145.308]
  MoveL 346 to (-200.15, 281.78, -8.41) mm, rotated rx -174.06 ry -29.54 rz -11.91 deg; joints [4.416, -43.13, 98.586, -77.089, 61.955, 145.307]
  MoveL 347 to (-206.05, 281.78, -11.57) mm, rotated rx -174.06 ry -29.54 rz -11.91 deg; joints [4.2, -43.001, 98.631, -77.344, 61.797, 145.469]
  MoveL 348 to (-201.08, 281.78, -20.25) mm, rotated rx -174.06 ry -29.54 rz -11.91 deg; joints [4.384, -42.571, 98.594, -77.409, 61.813, 145.93]
  MoveL 349 to (-201.08, 278.61, -20.25) mm, rotated rx -174.06 ry -29.54 rz -11.91 deg; joints [4.393, -42.721, 98.902, -77.485, 61.783, 146.106]
  MoveL 350 to (-206.05, 278.61, -11.57) mm, rotated rx -174.06 ry -29.54 rz -11.91 deg; joints [4.209, -43.153, 98.94, -77.42, 61.768, 145.644]
  MoveL 351 to (-200.15, 278.61, -8.41) mm, rotated rx -174.06 ry -29.54 rz -11.91 deg; joints [4.425, -43.282, 98.894, -77.164, 61.926, 145.481]
  MoveL 352 to (-197.85, 278.61, -8.4) mm, rotated rx -174.06 ry -29.54 rz -11.91 deg; joints [4.51, -43.274, 98.876, -77.094, 61.975, 145.482]
  MoveL 353 to (-197.85, 278.61, -4.14) mm, rotated rx -174.06 ry -29.54 rz -11.91 deg; joints [4.509, -43.476, 98.873, -76.988, 62.02, 145.256]
  Set speed (38.1 mm/s)
  MoveL 354 to (-197.89, 278.61, -3.98) mm, rotated rx -174.06 ry -29.54 rz -11.91 deg; joints [4.508, -43.483, 98.873, -76.986, 62.021, 145.247]
  MoveL 355 to (-198.05, 278.29, -3.7) mm, rotated rx -174.06 ry -29.54 rz -11.91 deg; joints [4.503, -43.512, 98.905, -76.991, 62.017, 145.25]
  Set speed (76.2 mm/s)
  MoveL 356 to (-198.05, 275.75, -3.7) mm, rotated rx -174.06 ry -29.54 rz -11.91 deg; joints [4.51, -43.634, 99.151, -77.05, 61.994, 145.388]
  Set speed (38.1 mm/s)
  MoveL 357 to (-197.89, 275.43, -3.98) mm, rotated rx -174.06 ry -29.54 rz -11.91 deg; joints [4.517, -43.636, 99.181, -77.059, 61.991, 145.42]
  MoveL 358 to (-197.85, 275.43, -4.14) mm, rotated rx -174.06 ry -29.54 rz -11.91 deg; joints [4.519, -43.628, 99.181, -77.062, 61.99, 145.428]
  Set speed (76.2 mm/s)
  MoveL 359 to (-197.85, 275.43, -8.4) mm, rotated rx -174.06 ry -29.54 rz -11.91 deg; joints [4.519, -43.426, 99.184, -77.168, 61.945, 145.656]
  MoveL 360 to (-200.15, 275.43, -8.41) mm, rotated rx -174.06 ry -29.54 rz -11.91 deg; joints [4.434, -43.434, 99.202, -77.238, 61.896, 145.654]
  MoveL 361 to (-206.05, 275.43, -11.57) mm, rotated rx -174.06 ry -29.54 rz -11.91 deg; joints [4.217, -43.304, 99.247, -77.495, 61.739, 145.818]
  MoveL 362 to (-201.08, 275.43, -20.25) mm, rotated rx -174.06 ry -29.54 rz -11.91 deg; joints [4.402, -42.871, 99.21, -77.56, 61.754, 146.282]
  MoveL 363 to (-201.08, 272.26, -20.25) mm, rotated rx -174.06 ry -29.54 rz -11.91 deg; joints [4.412, -43.021, 99.517, -77.636, 61.725, 146.457]
  MoveL 364 to (-206.05, 272.26, -11.57) mm, rotated rx -174.06 ry -29.54 rz -11.91 deg; joints [4.226, -43.454, 99.554, -77.57, 61.71, 145.992]
  MoveL 365 to (-200.15, 272.26, -8.41) mm, rotated rx -174.06 ry -29.54 rz -11.91 deg; joints [4.444, -43.585, 99.508, -77.312, 61.867, 145.828]
  MoveL 366 to (-197.85, 272.26, -8.4) mm, rotated rx -174.06 ry -29.54 rz -11.91 deg; joints [4.529, -43.577, 99.49, -77.242, 61.916, 145.829]
  MoveL 367 to (-197.85, 272.26, -4.14) mm, rotated rx -174.06 ry -29.54 rz -11.91 deg; joints [4.528, -43.78, 99.487, -77.135, 61.961, 145.601]
  Set speed (38.1 mm/s)
  MoveL 368 to (-197.89, 272.26, -3.98) mm, rotated rx -174.06 ry -29.54 rz -11.91 deg; joints [4.527, -43.787, 99.487, -77.132, 61.962, 145.592]
  MoveL 369 to (-198.05, 271.94, -3.7) mm, rotated rx -174.06 ry -29.54 rz -11.91 deg; joints [4.522, -43.816, 99.519, -77.138, 61.958, 145.595]
  Set speed (76.2 mm/s)
  MoveL 370 to (-198.05, 269.4, -3.7) mm, rotated rx -174.06 ry -29.54 rz -11.91 deg; joints [4.529, -43.937, 99.764, -77.196, 61.935, 145.732]
  Set speed (38.1 mm/s)
  MoveL 371 to (-197.89, 269.08, -3.98) mm, rotated rx -174.06 ry -29.54 rz -11.91 deg; joints [4.536, -43.939, 99.793, -77.205, 61.933, 145.764]
  MoveL 372 to (-197.85, 269.08, -4.14) mm, rotated rx -174.06 ry -29.54 rz -11.91 deg; joints [4.538, -43.931, 99.793, -77.208, 61.932, 145.773]
  Set speed (76.2 mm/s)
  MoveL 373 to (-197.85, 269.08, -8.4) mm, rotated rx -174.06 ry -29.54 rz -11.91 deg; joints [4.538, -43.728, 99.796, -77.315, 61.887, 146.001]
  MoveL 374 to (-200.15, 269.08, -8.41) mm, rotated rx -174.06 ry -29.54 rz -11.91 deg; joints [4.453, -43.736, 99.814, -77.386, 61.838, 146.001]
  MoveL 375 to (-206.05, 269.08, -11.57) mm, rotated rx -174.06 ry -29.54 rz -11.91 deg; joints [4.235, -43.605, 99.86, -77.645, 61.682, 146.166]
  MoveL 376 to (-201.08, 269.08, -20.25) mm, rotated rx -174.06 ry -29.54 rz -11.91 deg; joints [4.421, -43.17, 99.822, -77.711, 61.697, 146.632]
  MoveL 377 to (-201.08, 265.91, -20.25) mm, rotated rx -174.06 ry -29.54 rz -11.91 deg; joints [4.43, -43.319, 100.127, -77.786, 61.669, 146.806]
  MoveL 378 to (-206.05, 265.91, -11.57) mm, rotated rx -174.06 ry -29.54 rz -11.91 deg; joints [4.244, -43.755, 100.165, -77.72, 61.653, 146.339]
  MoveL 379 to (-200.15, 265.91, -8.41) mm, rotated rx -174.06 ry -29.54 rz -11.91 deg; joints [4.462, -43.886, 100.119, -77.459, 61.809, 146.173]
  MoveL 380 to (-197.85, 265.91, -8.4) mm, rotated rx -174.06 ry -29.54 rz -11.91 deg; joints [4.548, -43.878, 100.101, -77.388, 61.858, 146.174]
  MoveL 381 to (-197.85, 265.91, -4.14) mm, rotated rx -174.06 ry -29.54 rz -11.91 deg; joints [4.547, -44.082, 100.098, -77.281, 61.903, 145.945]
  Set speed (38.1 mm/s)
  MoveL 382 to (-197.89, 265.91, -3.98) mm, rotated rx -174.06 ry -29.54 rz -11.91 deg; joints [4.546, -44.09, 100.098, -77.278, 61.904, 145.936]
  MoveL 383 to (-198.05, 265.59, -3.7) mm, rotated rx -174.06 ry -29.54 rz -11.91 deg; joints [4.541, -44.118, 100.13, -77.284, 61.901, 145.938]
  Set speed (76.2 mm/s)
  MoveL 384 to (-198.05, 263.05, -3.7) mm, rotated rx -174.06 ry -29.54 rz -11.91 deg; joints [4.548, -44.239, 100.373, -77.342, 61.878, 146.075]
  Set speed (38.1 mm/s)
  MoveL 385 to (-197.89, 262.73, -3.98) mm, rotated rx -174.06 ry -29.54 rz -11.91 deg; joints [4.555, -44.24, 100.403, -77.351, 61.875, 146.107]
  MoveL 386 to (-197.85, 262.73, -4.14) mm, rotated rx -174.06 ry -29.54 rz -11.91 deg; joints [4.557, -44.232, 100.402, -77.354, 61.875, 146.116]
  Set speed (76.2 mm/s)
  MoveL 387 to (-197.85, 262.73, -8.4) mm, rotated rx -174.06 ry -29.54 rz -11.91 deg; joints [4.558, -44.028, 100.406, -77.462, 61.83, 146.346]
  MoveL 388 to (-200.15, 262.73, -8.41) mm, rotated rx -174.06 ry -29.54 rz -11.91 deg; joints [4.472, -44.036, 100.423, -77.533, 61.781, 146.345]
  MoveL 389 to (-206.05, 262.73, -11.57) mm, rotated rx -174.06 ry -29.54 rz -11.91 deg; joints [4.253, -43.904, 100.469, -77.794, 61.625, 146.512]
  MoveL 390 to (-201.08, 262.73, -20.25) mm, rotated rx -174.06 ry -29.54 rz -11.91 deg; joints [4.44, -43.467, 100.431, -77.861, 61.641, 146.981]
  MoveL 391 to (-201.08, 259.56, -20.25) mm, rotated rx -174.06 ry -29.54 rz -11.91 deg; joints [4.449, -43.615, 100.735, -77.936, 61.613, 147.155]
  MoveL 392 to (-206.05, 259.56, -11.57) mm, rotated rx -174.06 ry -29.54 rz -11.91 deg; joints [4.262, -44.053, 100.772, -77.869, 61.598, 146.685]
  MoveL 393 to (-200.15, 259.56, -8.41) mm, rotated rx -174.06 ry -29.54 rz -11.91 deg; joints [4.481, -44.185, 100.727, -77.606, 61.753, 146.517]
  MoveL 394 to (-197.85, 259.56, -8.4) mm, rotated rx -174.06 ry -29.54 rz -11.91 deg; joints [4.567, -44.177, 100.709, -77.535, 61.802, 146.518]
  MoveL 395 to (-197.85, 259.56, -4.14) mm, rotated rx -174.06 ry -29.54 rz -11.91 deg; joints [4.566, -44.382, 100.706, -77.426, 61.846, 146.287]
  Set speed (38.1 mm/s)
  MoveL 396 to (-197.89, 259.56, -3.98) mm, rotated rx -174.06 ry -29.54 rz -11.91 deg; joints [4.565, -44.39, 100.706, -77.424, 61.847, 146.278]
  MoveL 397 to (-198.05, 259.24, -3.7) mm, rotated rx -174.06 ry -29.54 rz -11.91 deg; joints [4.56, -44.419, 100.737, -77.429, 61.844, 146.28]
  Set speed (76.2 mm/s)
  MoveL 398 to (-198.05, 256.7, -3.7) mm, rotated rx -174.06 ry -29.54 rz -11.91 deg; joints [4.567, -44.539, 100.979, -77.487, 61.821, 146.417]
  Set speed (38.1 mm/s)
  MoveL 399 to (-197.89, 256.38, -3.98) mm, rotated rx -174.06 ry -29.54 rz -11.91 deg; joints [4.574, -44.54, 101.008, -77.496, 61.819, 146.449]
  MoveL 400 to (-197.85, 256.38, -4.14) mm, rotated rx -174.06 ry -29.54 rz -11.91 deg; joints [4.576, -44.532, 101.008, -77.499, 61.818, 146.458]
  Set speed (76.2 mm/s)
  MoveL 401 to (-197.85, 256.38, -8.4) mm, rotated rx -174.06 ry -29.54 rz -11.91 deg; joints [4.577, -44.327, 101.011, -77.608, 61.774, 146.689]
  MoveL 402 to (-200.15, 256.38, -8.41) mm, rotated rx -174.06 ry -29.54 rz -11.91 deg; joints [4.491, -44.334, 101.029, -77.679, 61.725, 146.688]
  MoveL 403 to (-206.05, 256.38, -11.57) mm, rotated rx -174.06 ry -29.54 rz -11.91 deg; joints [4.271, -44.202, 101.075, -77.943, 61.57, 146.857]
  MoveL 404 to (-201.08, 256.38, -20.25) mm, rotated rx -174.06 ry -29.54 rz -11.91 deg; joints [4.458, -43.763, 101.037, -78.01, 61.586, 147.328]
  MoveL 405 to (-201.08, 253.21, -20.25) mm, rotated rx -174.06 ry -29.54 rz -11.91 deg; joints [4.468, -43.91, 101.339, -78.085, 61.559, 147.501]
  MoveL 406 to (-206.05, 253.21, -11.57) mm, rotated rx -174.06 ry -29.54 rz -11.91 deg; joints [4.28, -44.35, 101.376, -78.018, 61.543, 147.029]
  MoveL 407 to (-200.15, 253.21, -8.41) mm, rotated rx -174.06 ry -29.54 rz -11.91 deg; joints [4.5, -44.483, 101.331, -77.753, 61.698, 146.86]
  MoveL 408 to (-197.85, 253.21, -8.4) mm, rotated rx -174.06 ry -29.54 rz -11.91 deg; joints [4.587, -44.475, 101.313, -77.681, 61.746, 146.86]
  MoveL 409 to (-197.85, 253.21, -4.14) mm, rotated rx -174.06 ry -29.54 rz -11.91 deg; joints [4.586, -44.681, 101.31, -77.571, 61.791, 146.628]
  Set speed (38.1 mm/s)
  MoveL 410 to (-197.89, 253.21, -3.98) mm, rotated rx -174.06 ry -29.54 rz -11.91 deg; joints [4.584, -44.689, 101.31, -77.569, 61.791, 146.619]
  MoveL 411 to (-198.05, 252.89, -3.7) mm, rotated rx -174.06 ry -29.54 rz -11.91 deg; joints [4.579, -44.718, 101.341, -77.574, 61.788, 146.621]
  Set speed (76.2 mm/s)
  MoveL 412 to (-198.05, 250.35, -3.7) mm, rotated rx -174.06 ry -29.54 rz -11.91 deg; joints [4.587, -44.837, 101.582, -77.631, 61.766, 146.757]
  Set speed (38.1 mm/s)
  MoveL 413 to (-197.89, 250.03, -3.98) mm, rotated rx -174.06 ry -29.54 rz -11.91 deg; joints [4.594, -44.838, 101.611, -77.641, 61.764, 146.789]
  MoveL 414 to (-197.85, 250.03, -4.14) mm, rotated rx -174.06 ry -29.54 rz -11.91 deg; joints [4.595, -44.83, 101.611, -77.644, 61.763, 146.798]
  Set speed (76.2 mm/s)
  MoveL 415 to (-197.85, 250.03, -8.4) mm, rotated rx -174.06 ry -29.54 rz -11.91 deg; joints [4.596, -44.624, 101.614, -77.753, 61.719, 147.031]
  MoveL 416 to (-200.15, 250.03, -8.41) mm, rotated rx -174.06 ry -29.54 rz -11.91 deg; joints [4.51, -44.631, 101.632, -77.826, 61.671, 147.03]
  MoveL 417 to (-206.05, 250.03, -11.57) mm, rotated rx -174.06 ry -29.54 rz -11.91 deg; joints [4.289, -44.498, 101.677, -78.092, 61.516, 147.201]
  MoveL 418 to (-201.08, 250.03, -20.25) mm, rotated rx -174.06 ry -29.54 rz -11.91 deg; joints [4.477, -44.057, 101.64, -78.159, 61.532, 147.674]
  MoveL 419 to (-201.08, 246.86, -20.25) mm, rotated rx -174.06 ry -29.54 rz -11.91 deg; joints [4.487, -44.203, 101.94, -78.233, 61.506, 147.847]
  MoveL 420 to (-206.05, 246.86, -11.57) mm, rotated rx -174.06 ry -29.54 rz -11.91 deg; joints [4.298, -44.646, 101.978, -78.166, 61.49, 147.372]
  MoveL 421 to (-200.15, 246.86, -8.41) mm, rotated rx -174.06 ry -29.54 rz -11.91 deg; joints [4.519, -44.779, 101.932, -77.898, 61.644, 147.201]
  MoveL 422 to (-197.85, 246.86, -8.4) mm, rotated rx -174.06 ry -29.54 rz -11.91 deg; joints [4.606, -44.772, 101.915, -77.826, 61.692, 147.201]
  MoveL 423 to (-197.85, 246.86, -4.14) mm, rotated rx -174.06 ry -29.54 rz -11.91 deg; joints [4.605, -44.979, 101.911, -77.716, 61.736, 146.967]
  Set speed (38.1 mm/s)
  MoveL 424 to (-197.89, 246.86, -3.98) mm, rotated rx -174.06 ry -29.54 rz -11.91 deg; joints [4.604, -44.987, 101.912, -77.713, 61.737, 146.959]
  MoveL 425 to (-198.05, 246.54, -3.7) mm, rotated rx -174.06 ry -29.54 rz -11.91 deg; joints [4.599, -45.015, 101.943, -77.718, 61.734, 146.961]
  Set speed (76.2 mm/s)
  MoveL 426 to (-198.05, 244, -3.7) mm, rotated rx -174.06 ry -29.54 rz -11.91 deg; joints [4.606, -45.134, 102.182, -77.776, 61.712, 147.096]
  Set speed (38.1 mm/s)
  MoveL 427 to (-197.89, 243.69, -3.98) mm, rotated rx -174.06 ry -29.54 rz -11.91 deg; joints [4.613, -45.135, 102.211, -77.785, 61.71, 147.128]
  MoveL 428 to (-197.85, 243.69, -4.14) mm, rotated rx -174.06 ry -29.54 rz -11.91 deg; joints [4.615, -45.127, 102.211, -77.788, 61.709, 147.137]
  Set speed (76.2 mm/s)
  MoveL 429 to (-197.85, 243.69, -8.4) mm, rotated rx -174.06 ry -29.54 rz -11.91 deg; joints [4.616, -44.919, 102.214, -77.898, 61.665, 147.371]
  MoveL 430 to (-200.15, 243.69, -8.41) mm, rotated rx -174.06 ry -29.54 rz -11.91 deg; joints [4.529, -44.927, 102.232, -77.971, 61.617, 147.371]
  MoveL 431 to (-206.05, 243.69, -11.57) mm, rotated rx -174.06 ry -29.54 rz -11.91 deg; joints [4.308, -44.793, 102.277, -78.24, 61.463, 147.543]
  MoveL 432 to (-201.08, 243.69, -20.25) mm, rotated rx -174.06 ry -29.54 rz -11.91 deg; joints [4.496, -44.349, 102.24, -78.307, 61.48, 148.019]
  MoveL 433 to (-201.08, 240.51, -20.25) mm, rotated rx -174.06 ry -29.54 rz -11.91 deg; joints [4.506, -44.495, 102.539, -78.381, 61.454, 148.191]
  MoveL 434 to (-206.05, 240.51, -11.57) mm, rotated rx -174.06 ry -29.54 rz -11.91 deg; joints [4.317, -44.94, 102.576, -78.313, 61.437, 147.713]
  MoveL 435 to (-200.15, 240.51, -8.41) mm, rotated rx -174.06 ry -29.54 rz -11.91 deg; joints [4.539, -45.074, 102.531, -78.044, 61.591, 147.541]
  MoveL 436 to (-197.85, 240.51, -8.4) mm, rotated rx -174.06 ry -29.54 rz -11.91 deg; joints [4.626, -45.066, 102.513, -77.97, 61.639, 147.541]
  MoveL 437 to (-197.85, 240.51, -4.14) mm, rotated rx -174.06 ry -29.54 rz -11.91 deg; joints [4.625, -45.275, 102.51, -77.859, 61.683, 147.306]
  Set speed (38.1 mm/s)
  MoveL 438 to (-197.89, 240.51, -3.98) mm, rotated rx -174.06 ry -29.54 rz -11.91 deg; joints [4.623, -45.283, 102.51, -77.857, 61.683, 147.297]
  MoveL 439 to (-198.05, 240.19, -3.7) mm, rotated rx -174.06 ry -29.54 rz -11.91 deg; joints [4.618, -45.311, 102.541, -77.862, 61.68, 147.298]
  Set speed (76.2 mm/s)
  MoveL 440 to (-198.05, 237.65, -3.7) mm, rotated rx -174.06 ry -29.54 rz -11.91 deg; joints [4.626, -45.429, 102.779, -77.919, 61.659, 147.433]
  Set speed (38.1 mm/s)
  MoveL 441 to (-197.89, 237.34, -3.98) mm, rotated rx -174.06 ry -29.54 rz -11.91 deg; joints [4.633, -45.43, 102.808, -77.928, 61.657, 147.465]
  MoveL 442 to (-197.85, 237.34, -4.14) mm, rotated rx -174.06 ry -29.54 rz -11.91 deg; joints [4.635, -45.422, 102.808, -77.931, 61.656, 147.474]
  Set speed (76.2 mm/s)
  MoveL 443 to (-197.85, 237.34, -8.4) mm, rotated rx -174.06 ry -29.54 rz -11.91 deg; joints [4.636, -45.213, 102.811, -78.042, 61.612, 147.71]
  MoveL 444 to (-200.15, 237.34, -8.41) mm, rotated rx -174.06 ry -29.54 rz -11.91 deg; joints [4.548, -45.221, 102.828, -78.116, 61.565, 147.71]
  MoveL 445 to (-206.05, 237.34, -11.57) mm, rotated rx -174.06 ry -29.54 rz -11.91 deg; joints [4.326, -45.086, 102.874, -78.387, 61.412, 147.883]
  MoveL 446 to (-201.08, 237.34, -20.25) mm, rotated rx -174.06 ry -29.54 rz -11.91 deg; joints [4.516, -44.64, 102.837, -78.455, 61.428, 148.362]
  MoveL 447 to (-201.08, 234.16, -20.25) mm, rotated rx -174.06 ry -29.54 rz -11.91 deg; joints [4.525, -44.785, 103.134, -78.529, 61.403, 148.534]
  MoveL 448 to (-206.05, 234.16, -11.57) mm, rotated rx -174.06 ry -29.54 rz -11.91 deg; joints [4.335, -45.232, 103.171, -78.46, 61.386, 148.053]
  MoveL 449 to (-200.15, 234.16, -8.41) mm, rotated rx -174.06 ry -29.54 rz -11.91 deg; joints [4.558, -45.367, 103.126, -78.188, 61.539, 147.879]
  MoveL 450 to (-197.85, 234.16, -8.4) mm, rotated rx -174.06 ry -29.54 rz -11.91 deg; joints [4.646, -45.359, 103.108, -78.114, 61.586, 147.879]
  MoveL 451 to (-197.85, 234.16, -4.14) mm, rotated rx -174.06 ry -29.54 rz -11.91 deg; joints [4.645, -45.569, 103.105, -78.003, 61.63, 147.642]
  Set speed (38.1 mm/s)
  MoveL 452 to (-197.89, 234.16, -3.98) mm, rotated rx -174.06 ry -29.54 rz -11.91 deg; joints [4.643, -45.577, 103.105, -78, 61.631, 147.634]
  MoveL 453 to (-198.05, 233.84, -3.7) mm, rotated rx -174.06 ry -29.54 rz -11.91 deg; joints [4.638, -45.606, 103.136, -78.005, 61.628, 147.635]
  Set speed (76.2 mm/s)
  MoveL 454 to (-198.05, 231.3, -3.7) mm, rotated rx -174.06 ry -29.54 rz -11.91 deg; joints [4.646, -45.723, 103.373, -78.062, 61.607, 147.769]
  Set speed (38.1 mm/s)
  MoveL 455 to (-197.89, 230.99, -3.98) mm, rotated rx -174.06 ry -29.54 rz -11.91 deg; joints [4.653, -45.724, 103.402, -78.071, 61.605, 147.801]
  MoveL 456 to (-197.85, 230.99, -4.14) mm, rotated rx -174.06 ry -29.54 rz -11.91 deg; joints [4.655, -45.716, 103.401, -78.074, 61.604, 147.81]
  Set speed (76.2 mm/s)
  MoveL 457 to (-197.85, 230.99, -8.4) mm, rotated rx -174.06 ry -29.54 rz -11.91 deg; joints [4.656, -45.506, 103.405, -78.186, 61.561, 148.048]
  MoveL 458 to (-200.15, 230.99, -8.41) mm, rotated rx -174.06 ry -29.54 rz -11.91 deg; joints [4.568, -45.513, 103.422, -78.261, 61.513, 148.048]
  MoveL 459 to (-206.05, 230.99, -11.57) mm, rotated rx -174.06 ry -29.54 rz -11.91 deg; joints [4.345, -45.377, 103.467, -78.534, 61.361, 148.223]
  MoveL 460 to (-201.08, 230.99, -20.25) mm, rotated rx -174.06 ry -29.54 rz -11.91 deg; joints [4.535, -44.929, 103.43, -78.602, 61.377, 148.705]
  MoveL 461 to (-201.08, 227.81, -20.25) mm, rotated rx -174.06 ry -29.54 rz -11.91 deg; joints [4.545, -45.073, 103.726, -78.676, 61.353, 148.875]
  MoveL 462 to (-206.05, 227.81, -11.57) mm, rotated rx -174.06 ry -29.54 rz -11.91 deg; joints [4.354, -45.523, 103.763, -78.607, 61.336, 148.392]
  MoveL 463 to (-200.15, 227.81, -8.41) mm, rotated rx -174.06 ry -29.54 rz -11.91 deg; joints [4.578, -45.659, 103.718, -78.333, 61.488, 148.216]
  MoveL 464 to (-197.85, 227.81, -8.4) mm, rotated rx -174.06 ry -29.54 rz -11.91 deg; joints [4.666, -45.651, 103.7, -78.258, 61.535, 148.216]
  MoveL 465 to (-197.85, 227.81, -4.14) mm, rotated rx -174.06 ry -29.54 rz -11.91 deg; joints [4.665, -45.862, 103.697, -78.145, 61.579, 147.978]
  Set speed (38.1 mm/s)
  MoveL 466 to (-197.89, 227.81, -3.98) mm, rotated rx -174.06 ry -29.54 rz -11.91 deg; joints [4.663, -45.87, 103.697, -78.142, 61.579, 147.969]
  MoveL 467 to (-198.05, 227.49, -3.7) mm, rotated rx -174.06 ry -29.54 rz -11.91 deg; joints [4.658, -45.899, 103.728, -78.147, 61.576, 147.97]
  Set speed (76.2 mm/s)
  MoveL 468 to (-198.05, 224.95, -3.7) mm, rotated rx -174.06 ry -29.54 rz -11.91 deg; joints [4.666, -46.015, 103.964, -78.204, 61.556, 148.104]
  Set speed (38.1 mm/s)
  MoveL 469 to (-197.89, 224.64, -3.98) mm, rotated rx -174.06 ry -29.54 rz -11.91 deg; joints [4.673, -46.016, 103.992, -78.213, 61.554, 148.136]
  MoveL 470 to (-197.85, 224.64, -4.14) mm, rotated rx -174.06 ry -29.54 rz -11.91 deg; joints [4.675, -46.008, 103.992, -78.216, 61.553, 148.145]
  Set speed (76.2 mm/s)
  MoveL 471 to (-197.85, 224.64, -8.4) mm, rotated rx -174.06 ry -29.54 rz -11.91 deg; joints [4.676, -45.797, 103.995, -78.33, 61.51, 148.384]
  MoveL 472 to (-200.15, 224.64, -8.41) mm, rotated rx -174.06 ry -29.54 rz -11.91 deg; joints [4.588, -45.804, 104.013, -78.404, 61.463, 148.384]
  MoveL 473 to (-206.05, 224.64, -11.57) mm, rotated rx -174.06 ry -29.54 rz -11.91 deg; joints [4.363, -45.668, 104.058, -78.68, 61.311, 148.561]
  MoveL 474 to (-201.08, 224.64, -20.25) mm, rotated rx -174.06 ry -29.54 rz -11.91 deg; joints [4.555, -45.217, 104.021, -78.749, 61.328, 149.045]
  MoveL 475 to (-201.08, 221.46, -20.25) mm, rotated rx -174.06 ry -29.54 rz -11.91 deg; joints [4.565, -45.36, 104.316, -78.822, 61.304, 149.215]
  MoveL 476 to (-206.05, 221.46, -11.57) mm, rotated rx -174.06 ry -29.54 rz -11.91 deg; joints [4.373, -45.812, 104.353, -78.753, 61.287, 148.73]
  MoveL 477 to (-200.15, 221.46, -8.41) mm, rotated rx -174.06 ry -29.54 rz -11.91 deg; joints [4.598, -45.949, 104.307, -78.476, 61.438, 148.552]
  MoveL 478 to (-197.85, 221.46, -8.4) mm, rotated rx -174.06 ry -29.54 rz -11.91 deg; joints [4.686, -45.942, 104.29, -78.401, 61.485, 148.552]
  MoveL 479 to (-197.85, 221.46, -4.14) mm, rotated rx -174.06 ry -29.54 rz -11.91 deg; joints [4.685, -46.153, 104.287, -78.287, 61.528, 148.312]
  Set speed (38.1 mm/s)
  MoveL 480 to (-197.89, 221.46, -3.98) mm, rotated rx -174.06 ry -29.54 rz -11.91 deg; joints [4.683, -46.161, 104.287, -78.284, 61.529, 148.303]
  MoveL 481 to (-198.05, 221.14, -3.7) mm, rotated rx -174.06 ry -29.54 rz -11.91 deg; joints [4.678, -46.19, 104.317, -78.289, 61.526, 148.304]
  Set speed (76.2 mm/s)
  MoveL 482 to (-198.05, 218.6, -3.7) mm, rotated rx -174.06 ry -29.54 rz -11.91 deg; joints [4.686, -46.306, 104.552, -78.346, 61.506, 148.438]
  Set speed (38.1 mm/s)
  MoveL 483 to (-197.89, 218.29, -3.98) mm, rotated rx -174.06 ry -29.54 rz -11.91 deg; joints [4.693, -46.307, 104.58, -78.355, 61.504, 148.47]
  MoveL 484 to (-197.85, 218.29, -4.14) mm, rotated rx -174.06 ry -29.54 rz -11.91 deg; joints [4.695, -46.299, 104.58, -78.358, 61.504, 148.479]
  Set speed (76.2 mm/s)
  MoveL 485 to (-197.85, 218.29, -8.4) mm, rotated rx -174.06 ry -29.54 rz -11.91 deg; joints [4.696, -46.086, 104.583, -78.472, 61.461, 148.719]
  MoveL 486 to (-200.15, 218.29, -8.41) mm, rotated rx -174.06 ry -29.54 rz -11.91 deg; joints [4.608, -46.094, 104.601, -78.548, 61.413, 148.72]
  MoveL 487 to (-206.05, 218.29, -11.57) mm, rotated rx -174.06 ry -29.54 rz -11.91 deg; joints [4.382, -45.956, 104.646, -78.826, 61.262, 148.898]
  MoveL 488 to (-201.08, 218.29, -20.25) mm, rotated rx -174.06 ry -29.54 rz -11.91 deg; joints [4.574, -45.503, 104.609, -78.895, 61.279, 149.385]
  MoveL 489 to (-201.08, 215.11, -20.25) mm, rotated rx -174.06 ry -29.54 rz -11.91 deg; joints [4.584, -45.646, 104.902, -78.968, 61.256, 149.555]
  MoveL 490 to (-206.05, 215.11, -11.57) mm, rotated rx -174.06 ry -29.54 rz -11.91 deg; joints [4.392, -46.1, 104.939, -78.898, 61.239, 149.066]
  MoveL 491 to (-200.15, 215.11, -8.41) mm, rotated rx -174.06 ry -29.54 rz -11.91 deg; joints [4.618, -46.238, 104.894, -78.619, 61.389, 148.887]
  MoveL 492 to (-197.85, 215.11, -8.4) mm, rotated rx -174.06 ry -29.54 rz -11.91 deg; joints [4.706, -46.23, 104.876, -78.543, 61.436, 148.886]
  MoveL 493 to (-197.85, 215.11, -4.14) mm, rotated rx -174.06 ry -29.54 rz -11.91 deg; joints [4.705, -46.443, 104.873, -78.429, 61.479, 148.645]
  Set speed (38.1 mm/s)
  MoveL 494 to (-197.89, 215.11, -3.98) mm, rotated rx -174.06 ry -29.54 rz -11.91 deg; joints [4.704, -46.452, 104.873, -78.426, 61.48, 148.636]
  MoveL 495 to (-198.05, 214.8, -3.7) mm, rotated rx -174.06 ry -29.54 rz -11.91 deg; joints [4.698, -46.48, 104.904, -78.431, 61.477, 148.637]
  Set speed (76.2 mm/s)
  MoveL 496 to (-198.05, 212.26, -3.7) mm, rotated rx -174.06 ry -29.54 rz -11.91 deg; joints [4.707, -46.596, 105.137, -78.487, 61.457, 148.77]
  Set speed (38.1 mm/s)
  MoveL 497 to (-197.89, 211.94, -3.98) mm, rotated rx -174.06 ry -29.54 rz -11.91 deg; joints [4.714, -46.596, 105.166, -78.497, 61.455, 148.802]
  MoveL 498 to (-197.85, 211.94, -4.14) mm, rotated rx -174.06 ry -29.54 rz -11.91 deg; joints [4.716, -46.588, 105.165, -78.499, 61.455, 148.811]
  Set speed (76.2 mm/s)
  MoveL 499 to (-197.85, 211.94, -8.4) mm, rotated rx -174.06 ry -29.54 rz -11.91 deg; joints [4.716, -46.374, 105.169, -78.614, 61.412, 149.053]
  MoveL 500 to (-200.15, 211.94, -8.41) mm, rotated rx -174.06 ry -29.54 rz -11.91 deg; joints [4.628, -46.382, 105.186, -78.691, 61.365, 149.054]
  MoveL 501 to (-206.05, 211.94, -11.57) mm, rotated rx -174.06 ry -29.54 rz -11.91 deg; joints [4.402, -46.243, 105.231, -78.971, 61.215, 149.234]
  MoveL 502 to (-201.08, 211.94, -20.25) mm, rotated rx -174.06 ry -29.54 rz -11.91 deg; joints [4.594, -45.788, 105.194, -79.041, 61.232, 149.724]
  MoveL 503 to (-201.08, 208.76, -20.25) mm, rotated rx -174.06 ry -29.54 rz -11.91 deg; joints [4.604, -45.93, 105.486, -79.114, 61.209, 149.892]
  MoveL 504 to (-206.05, 208.76, -11.57) mm, rotated rx -174.06 ry -29.54 rz -11.91 deg; joints [4.411, -46.387, 105.523, -79.043, 61.191, 149.401]
  MoveL 505 to (-200.15, 208.76, -8.41) mm, rotated rx -174.06 ry -29.54 rz -11.91 deg; joints [4.638, -46.526, 105.478, -78.762, 61.341, 149.22]
  MoveL 506 to (-197.85, 208.76, -8.4) mm, rotated rx -174.06 ry -29.54 rz -11.91 deg; joints [4.727, -46.518, 105.46, -78.685, 61.388, 149.22]
  MoveL 507 to (-197.85, 208.76, -4.14) mm, rotated rx -174.06 ry -29.54 rz -11.91 deg; joints [4.726, -46.732, 105.457, -78.57, 61.431, 148.977]
  Set speed (38.1 mm/s)
  MoveL 508 to (-197.89, 208.76, -3.98) mm, rotated rx -174.06 ry -29.54 rz -11.91 deg; joints [4.724, -46.74, 105.457, -78.567, 61.431, 148.968]
  MoveL 509 to (-198.05, 208.45, -3.7) mm, rotated rx -174.06 ry -29.54 rz -11.91 deg; joints [4.719, -46.769, 105.487, -78.572, 61.428, 148.969]
  Set speed (76.2 mm/s)
  MoveL 510 to (-198.05, 205.91, -3.7) mm, rotated rx -174.06 ry -29.54 rz -11.91 deg; joints [4.727, -46.884, 105.72, -78.628, 61.409, 149.101]
  Set speed (38.1 mm/s)
  MoveL 511 to (-197.89, 205.59, -3.98) mm, rotated rx -174.06 ry -29.54 rz -11.91 deg; joints [4.734, -46.884, 105.748, -78.637, 61.407, 149.133]
  MoveL 512 to (-197.85, 205.59, -4.14) mm, rotated rx -174.06 ry -29.54 rz -11.91 deg; joints [4.736, -46.876, 105.748, -78.64, 61.407, 149.142]
  Set speed (76.2 mm/s)
  MoveL 513 to (-197.85, 205.59, -8.4) mm, rotated rx -174.06 ry -29.54 rz -11.91 deg; joints [4.737, -46.661, 105.751, -78.756, 61.364, 149.386]
  MoveL 514 to (-200.15, 205.59, -8.41) mm, rotated rx -174.06 ry -29.54 rz -11.91 deg; joints [4.648, -46.669, 105.769, -78.833, 61.318, 149.387]
  MoveL 515 to (-206.05, 205.59, -11.57) mm, rotated rx -174.06 ry -29.54 rz -11.91 deg; joints [4.421, -46.529, 105.814, -79.115, 61.168, 149.568]
  MoveL 516 to (-201.08, 205.59, -20.25) mm, rotated rx -174.06 ry -29.54 rz -11.91 deg; joints [4.614, -46.072, 105.777, -79.186, 61.186, 150.061]
  MoveL 517 to (-201.08, 202.41, -20.25) mm, rotated rx -174.06 ry -29.54 rz -11.91 deg; joints [4.625, -46.213, 106.067, -79.258, 61.163, 150.229]
  MoveL 518 to (-206.05, 202.41, -11.57) mm, rotated rx -174.06 ry -29.54 rz -11.91 deg; joints [4.43, -46.672, 106.104, -79.187, 61.145, 149.735]
  MoveL 519 to (-200.15, 202.41, -8.41) mm, rotated rx -174.06 ry -29.54 rz -11.91 deg; joints [4.658, -46.812, 106.059, -78.904, 61.294, 149.553]
  MoveL 520 to (-197.85, 202.41, -8.4) mm, rotated rx -174.06 ry -29.54 rz -11.91 deg; joints [4.747, -46.804, 106.041, -78.827, 61.341, 149.552]
  MoveL 521 to (-197.85, 202.41, -4.14) mm, rotated rx -174.06 ry -29.54 rz -11.91 deg; joints [4.747, -47.019, 106.038, -78.71, 61.383, 149.307]
  Set speed (38.1 mm/s)
  MoveL 522 to (-197.89, 202.41, -3.98) mm, rotated rx -174.06 ry -29.54 rz -11.91 deg; joints [4.745, -47.028, 106.038, -78.707, 61.384, 149.298]
  MoveL 523 to (-198.05, 202.1, -3.7) mm, rotated rx -174.06 ry -29.54 rz -11.91 deg; joints [4.74, -47.056, 106.068, -78.712, 61.381, 149.299]
  Set speed (76.2 mm/s)
  MoveL 524 to (-198.05, 199.56, -3.7) mm, rotated rx -174.06 ry -29.54 rz -11.91 deg; joints [4.748, -47.171, 106.3, -78.768, 61.362, 149.431]
  Set speed (38.1 mm/s)
  MoveL 525 to (-197.89, 199.24, -3.98) mm, rotated rx -174.06 ry -29.54 rz -11.91 deg; joints [4.755, -47.171, 106.328, -78.777, 61.361, 149.463]
  MoveL 526 to (-197.85, 199.24, -4.14) mm, rotated rx -174.06 ry -29.54 rz -11.91 deg; joints [4.757, -47.163, 106.328, -78.78, 61.36, 149.472]
  Set speed (76.2 mm/s)
  MoveL 527 to (-197.85, 199.24, -8.4) mm, rotated rx -174.06 ry -29.54 rz -11.91 deg; joints [4.758, -46.947, 106.331, -78.897, 61.318, 149.717]
  MoveL 528 to (-200.15, 199.24, -8.41) mm, rotated rx -174.06 ry -29.54 rz -11.91 deg; joints [4.668, -46.954, 106.349, -78.975, 61.271, 149.718]
  MoveL 529 to (-206.05, 199.24, -11.57) mm, rotated rx -174.06 ry -29.54 rz -11.91 deg; joints [4.44, -46.814, 106.394, -79.259, 61.122, 149.901]
  MoveL 530 to (-201.08, 199.24, -20.25) mm, rotated rx -174.06 ry -29.54 rz -11.91 deg; joints [4.635, -46.354, 106.357, -79.331, 61.14, 150.397]
  MoveL 531 to (-201.08, 196.06, -20.25) mm, rotated rx -174.06 ry -29.54 rz -11.91 deg; joints [4.645, -46.494, 106.646, -79.403, 61.118, 150.565]
  MoveL 532 to (-206.05, 196.06, -11.57) mm, rotated rx -174.06 ry -29.54 rz -11.91 deg; joints [4.45, -46.956, 106.683, -79.331, 61.1, 150.068]
  MoveL 533 to (-200.15, 196.06, -8.41) mm, rotated rx -174.06 ry -29.54 rz -11.91 deg; joints [4.679, -47.097, 106.637, -79.045, 61.248, 149.884]
  MoveL 534 to (-197.85, 196.06, -8.4) mm, rotated rx -174.06 ry -29.54 rz -11.91 deg; joints [4.768, -47.089, 106.62, -78.968, 61.295, 149.883]
  MoveL 535 to (-197.85, 196.06, -4.14) mm, rotated rx -174.06 ry -29.54 rz -11.91 deg; joints [4.767, -47.305, 106.617, -78.85, 61.337, 149.637]
  Set speed (38.1 mm/s)
  MoveL 536 to (-197.89, 196.06, -3.98) mm, rotated rx -174.06 ry -29.54 rz -11.91 deg; joints [4.766, -47.314, 106.617, -78.847, 61.337, 149.627]
  MoveL 537 to (-198.05, 195.75, -3.7) mm, rotated rx -174.06 ry -29.54 rz -11.91 deg; joints [4.761, -47.342, 106.647, -78.852, 61.335, 149.628]
  Set speed (76.2 mm/s)
  MoveL 538 to (-198.05, 193.21, -3.7) mm, rotated rx -174.06 ry -29.54 rz -11.91 deg; joints [4.769, -47.456, 106.877, -78.908, 61.316, 149.759]
  Set speed (38.1 mm/s)
  MoveL 539 to (-197.89, 192.89, -3.98) mm, rotated rx -174.06 ry -29.54 rz -11.91 deg; joints [4.776, -47.456, 106.905, -78.917, 61.315, 149.791]
  MoveL 540 to (-197.85, 192.89, -4.14) mm, rotated rx -174.06 ry -29.54 rz -11.91 deg; joints [4.778, -47.448, 106.905, -78.92, 61.314, 149.801]
  Set speed (76.2 mm/s)
  MoveL 541 to (-197.85, 192.89, -8.4) mm, rotated rx -174.06 ry -29.54 rz -11.91 deg; joints [4.779, -47.231, 106.908, -79.038, 61.272, 150.048]
  MoveL 542 to (-199.6, 192.89, -8.41) mm, rotated rx -174.06 ry -29.54 rz -11.91 deg; joints [4.711, -47.236, 106.921, -79.097, 61.237, 150.049]
  MoveL 543 to (-206.05, 192.89, -11.57) mm, rotated rx -174.06 ry -29.54 rz -11.91 deg; joints [4.46, -47.097, 106.971, -79.403, 61.078, 150.234]
  MoveL 544 to (-201.08, 192.89, -20.25) mm, rotated rx -174.06 ry -29.54 rz -11.91 deg; joints [4.655, -46.634, 106.934, -79.475, 61.096, 150.732]
  MoveL 545 to (-201.08, 189.71, -20.25) mm, rotated rx -174.06 ry -29.54 rz -11.91 deg; joints [4.666, -46.774, 107.221, -79.547, 61.074, 150.899]
  MoveL 546 to (-206.05, 189.71, -11.57) mm, rotated rx -174.06 ry -29.54 rz -11.91 deg; joints [4.47, -47.238, 107.258, -79.475, 61.056, 150.399]
  MoveL 547 to (-199.6, 189.71, -8.41) mm, rotated rx -174.06 ry -29.54 rz -11.91 deg; joints [4.721, -47.378, 107.209, -79.167, 61.215, 150.213]
  MoveL 548 to (-197.85, 189.71, -8.4) mm, rotated rx -174.06 ry -29.54 rz -11.91 deg; joints [4.789, -47.372, 107.196, -79.108, 61.25, 150.212]
  MoveL 549 to (-197.85, 189.71, -4.14) mm, rotated rx -174.06 ry -29.54 rz -11.91 deg; joints [4.788, -47.59, 107.192, -78.99, 61.291, 149.965]
  MoveL 550 to (-197.85, 189.59, -3.66) mm, rotated rx -174.06 ry -29.54 rz -11.91 deg; joints [4.789, -47.62, 107.204, -78.979, 61.295, 149.943]
  MoveL 551 to (-197.85, 189.24, -3.31) mm, rotated rx -174.06 ry -29.54 rz -11.91 deg; joints [4.79, -47.653, 107.235, -78.977, 61.296, 149.941]
  MoveL 552 to (-197.85, 188.76, -3.19) mm, rotated rx -174.06 ry -29.54 rz -11.91 deg; joints [4.791, -47.681, 107.278, -78.984, 61.294, 149.958]
  MoveL 553 to (-197.85, 187.49, -3.19) mm, rotated rx -174.06 ry -29.54 rz -11.91 deg; joints [4.796, -47.738, 107.392, -79.012, 61.285, 150.024]
  MoveL 554 to (-197.85, 187.02, -3.31) mm, rotated rx -174.06 ry -29.54 rz -11.91 deg; joints [4.797, -47.753, 107.436, -79.026, 61.28, 150.056]
  MoveL 555 to (-197.85, 186.67, -3.66) mm, rotated rx -174.06 ry -29.54 rz -11.91 deg; joints [4.799, -47.751, 107.467, -79.043, 61.275, 150.094]
  MoveL 556 to (-197.85, 186.54, -4.14) mm, rotated rx -174.06 ry -29.54 rz -11.91 deg; joints [4.799, -47.732, 107.479, -79.059, 61.269, 150.128]
  MoveL 557 to (-197.85, 186.54, -8.4) mm, rotated rx -174.06 ry -29.54 rz -11.91 deg; joints [4.8, -47.513, 107.483, -79.178, 61.228, 150.377]
  MoveL 558 to (-199.6, 186.54, -8.41) mm, rotated rx -174.06 ry -29.54 rz -11.91 deg; joints [4.731, -47.519, 107.496, -79.238, 61.192, 150.378]
  MoveL 559 to (-206.05, 186.54, -11.57) mm, rotated rx -174.06 ry -29.54 rz -11.91 deg; joints [4.48, -47.379, 107.545, -79.546, 61.034, 150.564]
  MoveL 560 to (-201.08, 186.54, -20.25) mm, rotated rx -174.06 ry -29.54 rz -11.91 deg; joints [4.676, -46.914, 107.508, -79.618, 61.052, 151.066]
  MoveL 561 to (-201.08, 183.37, -20.25) mm, rotated rx -174.06 ry -29.54 rz -11.91 deg; joints [4.686, -47.053, 107.795, -79.69, 61.031, 151.232]
  MoveL 562 to (-206.05, 183.37, -11.57) mm, rotated rx -174.06 ry -29.54 rz -11.91 deg; joints [4.49, -47.519, 107.832, -79.617, 61.012, 150.73]
  MoveL 563 to (-199.6, 183.37, -8.41) mm, rotated rx -174.06 ry -29.54 rz -11.91 deg; joints [4.742, -47.66, 107.782, -79.308, 61.17, 150.542]
  MoveL 564 to (-197.85, 183.37, -8.4) mm, rotated rx -174.06 ry -29.54 rz -11.91 deg; joints [4.811, -47.654, 107.769, -79.248, 61.206, 150.541]
  MoveL 565 to (-197.85, 183.37, -4.14) mm, rotated rx -174.06 ry -29.54 rz -11.91 deg; joints [4.81, -47.873, 107.766, -79.128, 61.247, 150.292]
  MoveL 566 to (-197.85, 183.24, -3.66) mm, rotated rx -174.06 ry -29.54 rz -11.91 deg; joints [4.81, -47.904, 107.777, -79.118, 61.251, 150.27]
  MoveL 567 to (-197.85, 182.89, -3.31) mm, rotated rx -174.06 ry -29.54 rz -11.91 deg; joints [4.811, -47.937, 107.808, -79.116, 61.252, 150.268]
  MoveL 568 to (-197.85, 182.41, -3.19) mm, rotated rx -174.06 ry -29.54 rz -11.91 deg; joints [4.813, -47.965, 107.851, -79.122, 61.25, 150.285]
  MoveL 569 to (-197.85, 181.14, -3.19) mm, rotated rx -174.06 ry -29.54 rz -11.91 deg; joints [4.817, -48.021, 107.965, -79.15, 61.241, 150.35]
  MoveL 570 to (-197.85, 180.67, -3.31) mm, rotated rx -174.06 ry -29.54 rz -11.91 deg; joints [4.819, -48.036, 108.008, -79.164, 61.236, 150.382]
  MoveL 571 to (-197.85, 180.32, -3.66) mm, rotated rx -174.06 ry -29.54 rz -11.91 deg; joints [4.82, -48.033, 108.04, -79.181, 61.23, 150.42]
  MoveL 572 to (-197.85, 180.19, -4.14) mm, rotated rx -174.06 ry -29.54 rz -11.91 deg; joints [4.82, -48.015, 108.051, -79.198, 61.225, 150.455]
  MoveL 573 to (-197.85, 180.19, -8.4) mm, rotated rx -174.06 ry -29.54 rz -11.91 deg; joints [4.821, -47.795, 108.055, -79.317, 61.184, 150.705]
  MoveL 574 to (-199.6, 180.19, -8.41) mm, rotated rx -174.06 ry -29.54 rz -11.91 deg; joints [4.752, -47.801, 108.068, -79.378, 61.149, 150.706]
  MoveL 575 to (-206.05, 180.19, -11.57) mm, rotated rx -174.06 ry -29.54 rz -11.91 deg; joints [4.5, -47.659, 108.117, -79.689, 60.991, 150.894]
  MoveL 576 to (-201.08, 180.19, -20.25) mm, rotated rx -174.06 ry -29.54 rz -11.91 deg; joints [4.697, -47.192, 108.08, -79.761, 61.009, 151.399]
  MoveL 577 to (-201.08, 177.02, -20.25) mm, rotated rx -174.06 ry -29.54 rz -11.91 deg; joints [4.707, -47.33, 108.366, -79.833, 60.988, 151.565]
  MoveL 578 to (-206.05, 177.02, -11.57) mm, rotated rx -174.06 ry -29.54 rz -11.91 deg; joints [4.51, -47.799, 108.402, -79.76, 60.97, 151.059]
  MoveL 579 to (-199.6, 177.02, -8.41) mm, rotated rx -174.06 ry -29.54 rz -11.91 deg; joints [4.763, -47.941, 108.353, -79.447, 61.127, 150.87]
  MoveL 580 to (-197.85, 177.02, -8.4) mm, rotated rx -174.06 ry -29.54 rz -11.91 deg; joints [4.832, -47.935, 108.34, -79.387, 61.162, 150.868]
  MoveL 581 to (-197.85, 177.02, -4.14) mm, rotated rx -174.06 ry -29.54 rz -11.91 deg; joints [4.831, -48.156, 108.337, -79.267, 61.203, 150.617]
  MoveL 582 to (-197.85, 176.89, -3.66) mm, rotated rx -174.06 ry -29.54 rz -11.91 deg; joints [4.831, -48.186, 108.348, -79.256, 61.207, 150.596]
  MoveL 583 to (-197.85, 176.54, -3.31) mm, rotated rx -174.06 ry -29.54 rz -11.91 deg; joints [4.833, -48.219, 108.378, -79.254, 61.208, 150.593]
  MoveL 584 to (-197.85, 176.06, -3.19) mm, rotated rx -174.06 ry -29.54 rz -11.91 deg; joints [4.834, -48.247, 108.421, -79.26, 61.206, 150.61]
  MoveL 585 to (-197.85, 174.79, -3.19) mm, rotated rx -174.06 ry -29.54 rz -11.91 deg; joints [4.838, -48.303, 108.535, -79.288, 61.197, 150.675]
  MoveL 586 to (-197.85, 174.32, -3.31) mm, rotated rx -174.06 ry -29.54 rz -11.91 deg; joints [4.84, -48.318, 108.578, -79.302, 61.193, 150.707]
  MoveL 587 to (-197.85, 173.97, -3.66) mm, rotated rx -174.06 ry -29.54 rz -11.91 deg; joints [4.841, -48.315, 108.609, -79.319, 61.187, 150.745]
  MoveL 588 to (-197.85, 173.84, -4.14) mm, rotated rx -174.06 ry -29.54 rz -11.91 deg; joints [4.842, -48.296, 108.621, -79.336, 61.182, 150.78]
  MoveL 589 to (-197.85, 173.84, -8.4) mm, rotated rx -174.06 ry -29.54 rz -11.91 deg; joints [4.843, -48.075, 108.624, -79.456, 61.141, 151.032]
  MoveL 590 to (-199.6, 173.84, -8.41) mm, rotated rx -174.06 ry -29.54 rz -11.91 deg; joints [4.774, -48.081, 108.638, -79.517, 61.106, 151.033]
  MoveL 591 to (-206.05, 173.84, -11.57) mm, rotated rx -174.06 ry -29.54 rz -11.91 deg; joints [4.52, -47.939, 108.687, -79.831, 60.949, 151.223]
  MoveL 592 to (-201.08, 173.84, -20.25) mm, rotated rx -174.06 ry -29.54 rz -11.91 deg; joints [4.718, -47.468, 108.65, -79.904, 60.968, 151.73]
  MoveL 593 to (-201.08, 170.67, -20.25) mm, rotated rx -174.06 ry -29.54 rz -11.91 deg; joints [4.728, -47.606, 108.934, -79.975, 60.947, 151.896]
  MoveL 594 to (-206.05, 170.67, -11.57) mm, rotated rx -174.06 ry -29.54 rz -11.91 deg; joints [4.53, -48.078, 108.971, -79.901, 60.929, 151.387]
  MoveL 595 to (-199.6, 170.67, -8.41) mm, rotated rx -174.06 ry -29.54 rz -11.91 deg; joints [4.784, -48.221, 108.922, -79.587, 61.085, 151.196]
  MoveL 596 to (-197.85, 170.67, -8.4) mm, rotated rx -174.06 ry -29.54 rz -11.91 deg; joints [4.854, -48.215, 108.908, -79.525, 61.12, 151.195]
  MoveL 597 to (-197.85, 170.67, -4.14) mm, rotated rx -174.06 ry -29.54 rz -11.91 deg; joints [4.853, -48.436, 108.905, -79.404, 61.161, 150.942]
  Set speed (38.1 mm/s)
  MoveL 598 to (-197.89, 170.67, -3.98) mm, rotated rx -174.06 ry -29.54 rz -11.91 deg; joints [4.851, -48.445, 108.905, -79.401, 61.161, 150.933]
  MoveL 599 to (-198.05, 170.35, -3.7) mm, rotated rx -174.06 ry -29.54 rz -11.91 deg; joints [4.846, -48.474, 108.934, -79.406, 61.159, 150.933]
  Set speed (76.2 mm/s)
  MoveL 600 to (-198.05, 167.81, -3.7) mm, rotated rx -174.06 ry -29.54 rz -11.91 deg; joints [4.854, -48.586, 109.161, -79.461, 61.142, 151.062]
  Set speed (38.1 mm/s)
  MoveL 601 to (-197.89, 167.49, -3.98) mm, rotated rx -174.06 ry -29.54 rz -11.91 deg; joints [4.862, -48.585, 109.188, -79.47, 61.14, 151.095]
  MoveL 602 to (-197.85, 167.49, -4.14) mm, rotated rx -174.06 ry -29.54 rz -11.91 deg; joints [4.864, -48.576, 109.188, -79.473, 61.14, 151.104]
  Set speed (76.2 mm/s)
  MoveL 603 to (-197.85, 167.49, -8.4) mm, rotated rx -174.06 ry -29.54 rz -11.91 deg; joints [4.865, -48.354, 109.191, -79.595, 61.099, 151.357]
  MoveL 604 to (-199.6, 167.49, -8.41) mm, rotated rx -174.06 ry -29.54 rz -11.91 deg; joints [4.795, -48.36, 109.205, -79.656, 61.064, 151.359]
  MoveL 605 to (-206.05, 167.49, -11.57) mm, rotated rx -174.06 ry -29.54 rz -11.91 deg; joints [4.54, -48.217, 109.254, -79.972, 60.908, 151.551]
  MoveL 606 to (-201.08, 167.49, -20.25) mm, rotated rx -174.06 ry -29.54 rz -11.91 deg; joints [4.739, -47.744, 109.217, -80.046, 60.927, 152.061]
  MoveL 607 to (-201.08, 164.32, -20.25) mm, rotated rx -174.06 ry -29.54 rz -11.91 deg; joints [4.749, -47.881, 109.5, -80.117, 60.907, 152.226]
  MoveL 608 to (-206.05, 164.32, -11.57) mm, rotated rx -174.06 ry -29.54 rz -11.91 deg; joints [4.55, -48.355, 109.537, -80.043, 60.888, 151.714]
  MoveL 609 to (-199.6, 164.32, -8.41) mm, rotated rx -174.06 ry -29.54 rz -11.91 deg; joints [4.806, -48.499, 109.487, -79.725, 61.044, 151.522]
  MoveL 610 to (-197.85, 164.32, -8.4) mm, rotated rx -174.06 ry -29.54 rz -11.91 deg; joints [4.875, -48.493, 109.474, -79.664, 61.078, 151.52]
  MoveL 611 to (-197.85, 164.32, -4.14) mm, rotated rx -174.06 ry -29.54 rz -11.91 deg; joints [4.875, -48.716, 109.471, -79.542, 61.119, 151.266]
  Set speed (38.1 mm/s)
  MoveL 612 to (-197.89, 164.32, -3.98) mm, rotated rx -174.06 ry -29.54 rz -11.91 deg; joints [4.873, -48.725, 109.471, -79.538, 61.119, 151.256]
  MoveL 613 to (-198.05, 164, -3.7) mm, rotated rx -174.06 ry -29.54 rz -11.91 deg; joints [4.868, -48.753, 109.5, -79.543, 61.117, 151.256]
  Set speed (76.2 mm/s)
  MoveL 614 to (-198.05, 161.46, -3.7) mm, rotated rx -174.06 ry -29.54 rz -11.91 deg; joints [4.876, -48.865, 109.726, -79.598, 61.1, 151.385]
  Set speed (38.1 mm/s)
  MoveL 615 to (-197.89, 161.14, -3.98) mm, rotated rx -174.06 ry -29.54 rz -11.91 deg; joints [4.884, -48.864, 109.753, -79.607, 61.099, 151.417]
  MoveL 616 to (-197.85, 161.14, -4.14) mm, rotated rx -174.06 ry -29.54 rz -11.91 deg; joints [4.886, -48.855, 109.753, -79.61, 61.098, 151.427]
  Set speed (76.2 mm/s)
  MoveL 617 to (-197.85, 161.14, -8.4) mm, rotated rx -174.06 ry -29.54 rz -11.91 deg; joints [4.886, -48.632, 109.756, -79.733, 61.058, 151.682]
  MoveL 618 to (-199.6, 161.14, -8.41) mm, rotated rx -174.06 ry -29.54 rz -11.91 deg; joints [4.817, -48.638, 109.769, -79.794, 61.023, 151.684]
  MoveL 619 to (-206.05, 161.14, -11.57) mm, rotated rx -174.06 ry -29.54 rz -11.91 deg; joints [4.561, -48.493, 109.819, -80.113, 60.868, 151.877]
  MoveL 620 to (-201.08, 161.14, -20.25) mm, rotated rx -174.06 ry -29.54 rz -11.91 deg; joints [4.76, -48.018, 109.782, -80.187, 60.887, 152.391]
  MoveL 621 to (-201.08, 157.97, -20.25) mm, rotated rx -174.06 ry -29.54 rz -11.91 deg; joints [4.771, -48.154, 110.063, -80.258, 60.867, 152.555]
  MoveL 622 to (-206.05, 157.97, -11.57) mm, rotated rx -174.06 ry -29.54 rz -11.91 deg; joints [4.571, -48.631, 110.1, -80.183, 60.849, 152.04]
  MoveL 623 to (-199.6, 157.97, -8.41) mm, rotated rx -174.06 ry -29.54 rz -11.91 deg; joints [4.828, -48.776, 110.051, -79.863, 61.003, 151.846]
  MoveL 624 to (-197.85, 157.97, -8.4) mm, rotated rx -174.06 ry -29.54 rz -11.91 deg; joints [4.897, -48.77, 110.038, -79.801, 61.038, 151.844]
  MoveL 625 to (-197.85, 157.97, -4.14) mm, rotated rx -174.06 ry -29.54 rz -11.91 deg; joints [4.897, -48.995, 110.034, -79.678, 61.078, 151.588]
  Set speed (38.1 mm/s)
  MoveL 626 to (-197.89, 157.97, -3.98) mm, rotated rx -174.06 ry -29.54 rz -11.91 deg; joints [4.895, -49.003, 110.034, -79.675, 61.079, 151.579]
  MoveL 627 to (-198.05, 157.65, -3.7) mm, rotated rx -174.06 ry -29.54 rz -11.91 deg; joints [4.89, -49.032, 110.064, -79.68, 61.076, 151.578]
  Set speed (76.2 mm/s)
  MoveL 628 to (-198.05, 155.11, -3.7) mm, rotated rx -174.06 ry -29.54 rz -11.91 deg; joints [4.898, -49.143, 110.288, -79.734, 61.06, 151.707]
  Set speed (38.1 mm/s)
  MoveL 629 to (-197.89, 154.79, -3.98) mm, rotated rx -174.06 ry -29.54 rz -11.91 deg; joints [4.906, -49.142, 110.315, -79.743, 61.058, 151.739]
  MoveL 630 to (-197.85, 154.79, -4.14) mm, rotated rx -174.06 ry -29.54 rz -11.91 deg; joints [4.908, -49.133, 110.315, -79.746, 61.058, 151.749]
  Set speed (76.2 mm/s)
  MoveL 631 to (-197.85, 154.79, -8.4) mm, rotated rx -174.06 ry -29.54 rz -11.91 deg; joints [4.909, -48.908, 110.318, -79.87, 61.018, 152.006]
  MoveL 632 to (-199.6, 154.79, -8.41) mm, rotated rx -174.06 ry -29.54 rz -11.91 deg; joints [4.838, -48.914, 110.332, -79.932, 60.983, 152.008]
  MoveL 633 to (-206.05, 154.79, -11.57) mm, rotated rx -174.06 ry -29.54 rz -11.91 deg; joints [4.581, -48.769, 110.381, -80.253, 60.829, 152.203]
  MoveL 634 to (-201.08, 154.79, -20.25) mm, rotated rx -174.06 ry -29.54 rz -11.91 deg; joints [4.782, -48.291, 110.344, -80.328, 60.848, 152.719]
  MoveL 635 to (-201.08, 151.62, -20.25) mm, rotated rx -174.06 ry -29.54 rz -11.91 deg; joints [4.793, -48.426, 110.625, -80.399, 60.829, 152.883]
  MoveL 636 to (-206.05, 151.62, -11.57) mm, rotated rx -174.06 ry -29.54 rz -11.91 deg; joints [4.592, -48.906, 110.662, -80.323, 60.81, 152.365]
  MoveL 637 to (-199.6, 151.62, -8.41) mm, rotated rx -174.06 ry -29.54 rz -11.91 deg; joints [4.849, -49.052, 110.612, -80.001, 60.964, 152.169]
  MoveL 638 to (-197.85, 151.62, -8.4) mm, rotated rx -174.06 ry -29.54 rz -11.91 deg; joints [4.92, -49.046, 110.599, -79.938, 60.998, 152.167]
  MoveL 639 to (-197.85, 151.62, -4.14) mm, rotated rx -174.06 ry -29.54 rz -11.91 deg; joints [4.919, -49.272, 110.595, -79.814, 61.038, 151.91]
  Set speed (38.1 mm/s)
  MoveL 640 to (-197.89, 151.62, -3.98) mm, rotated rx -174.06 ry -29.54 rz -11.91 deg; joints [4.917, -49.28, 110.596, -79.811, 61.039, 151.9]
  MoveL 641 to (-198.05, 151.3, -3.7) mm, rotated rx -174.06 ry -29.54 rz -11.91 deg; joints [4.912, -49.309, 110.625, -79.816, 61.036, 151.899]
  Set speed (76.2 mm/s)
  MoveL 642 to (-198.05, 148.76, -3.7) mm, rotated rx -174.06 ry -29.54 rz -11.91 deg; joints [4.921, -49.42, 110.848, -79.87, 61.02, 152.028]
  Set speed (38.1 mm/s)
  MoveL 643 to (-197.89, 148.44, -3.98) mm, rotated rx -174.06 ry -29.54 rz -11.91 deg; joints [4.928, -49.419, 110.875, -79.879, 61.019, 152.06]
  MoveL 644 to (-197.85, 148.44, -4.14) mm, rotated rx -174.06 ry -29.54 rz -11.91 deg; joints [4.93, -49.41, 110.875, -79.882, 61.018, 152.07]
